	MoveL Offs(p0,623.8,790.0, 0), v100, z5, tool0;
	MoveL Offs(p0,621.6576000000002,788.0128000000002, 0), v100, z5, tool0;
	MoveL Offs(p0,619.9534,786.1551999999999, 0), v100, z5, tool0;
	MoveL Offs(p0,617.8928,783.7984, 0), v100, z5, tool0;
	MoveL Offs(p0,615.525,781.0, 0), v100, z5, tool0;
	MoveL Offs(p0,612.8992000000001,777.8176, 0), v100, z5, tool0;
	MoveL Offs(p0,610.0645999999999,774.3088, 0), v100, z5, tool0;
	MoveL Offs(p0,607.0704000000001,770.5312, 0), v100, z5, tool0;
	MoveL Offs(p0,603.9658,766.5424, 0), v100, z5, tool0;
	MoveL Offs(p0,600.8,762.4, 0), v100, z5, tool0;
	MoveL Offs(p0,596.1566,756.2386000000001, 0), v100, z5, tool0;
	MoveL Offs(p0,592.2368000000002,751.1248000000003, 0), v100, z5, tool0;
	MoveL Offs(p0,588.9361999999999,746.9541999999999, 0), v100, z5, tool0;
	MoveL Offs(p0,586.1504000000001,743.6224, 0), v100, z5, tool0;
	MoveL Offs(p0,583.775,741.025, 0), v100, z5, tool0;
	MoveL Offs(p0,581.7056,739.0576, 0), v100, z5, tool0;
	MoveL Offs(p0,579.8378,737.6157999999999, 0), v100, z5, tool0;
	MoveL Offs(p0,578.0672000000001,736.5952000000001, 0), v100, z5, tool0;
	MoveL Offs(p0,576.2894,735.8914000000001, 0), v100, z5, tool0;
	MoveL Offs(p0,574.4,735.4, 0), v100, z5, tool0;
	MoveL Offs(p0,566.3782000000001,733.9154000000001, 0), v100, z5, tool0;
	MoveL Offs(p0,559.1856000000001,732.8352000000002, 0), v100, z5, tool0;
	MoveL Offs(p0,552.5713999999999,732.1798000000001, 0), v100, z5, tool0;
	MoveL Offs(p0,546.2848,731.9696, 0), v100, z5, tool0;
	MoveL Offs(p0,540.075,732.225, 0), v100, z5, tool0;
	MoveL Offs(p0,533.6912,732.9664, 0), v100, z5, tool0;
	MoveL Offs(p0,526.8826,734.2142, 0), v100, z5, tool0;
	MoveL Offs(p0,519.3984,735.9888000000001, 0), v100, z5, tool0;
	MoveL Offs(p0,510.98780000000005,738.3106, 0), v100, z5, tool0;
	MoveL Offs(p0,501.4,741.2, 0), v100, z5, tool0;
	MoveL Offs(p0,496.9594000000001,742.5744000000001, 0), v100, z5, tool0;
	MoveL Offs(p0,492.63520000000017,743.8192000000001, 0), v100, z5, tool0;
	MoveL Offs(p0,488.4237999999999,744.9368, 0), v100, z5, tool0;
	MoveL Offs(p0,484.32159999999993,745.9296, 0), v100, z5, tool0;
	MoveL Offs(p0,480.325,746.8, 0), v100, z5, tool0;
	MoveL Offs(p0,476.4304,747.5504, 0), v100, z5, tool0;
	MoveL Offs(p0,472.63419999999996,748.1832, 0), v100, z5, tool0;
	MoveL Offs(p0,468.93280000000004,748.7008000000001, 0), v100, z5, tool0;
	MoveL Offs(p0,465.3226000000001,749.1056000000001, 0), v100, z5, tool0;
	MoveL Offs(p0,461.8,749.4, 0), v100, z5, tool0;
	MoveL Offs(p0,444.6,750.6, 0), v100, z5, tool0;
	MoveL Offs(p0,443.2,768.8, 0), v100, z5, tool0;
	MoveL Offs(p0,442.5474000000001,776.1014, 0), v100, z5, tool0;
	MoveL Offs(p0,441.5792000000001,784.0592000000003, 0), v100, z5, tool0;
	MoveL Offs(p0,440.3398,792.4538000000001, 0), v100, z5, tool0;
	MoveL Offs(p0,438.87360000000007,801.0656000000001, 0), v100, z5, tool0;
	MoveL Offs(p0,437.225,809.675, 0), v100, z5, tool0;
	MoveL Offs(p0,435.4384,818.0624, 0), v100, z5, tool0;
	MoveL Offs(p0,433.55820000000006,826.0082, 0), v100, z5, tool0;
	MoveL Offs(p0,431.62880000000007,833.2928000000002, 0), v100, z5, tool0;
	MoveL Offs(p0,429.6946,839.6966, 0), v100, z5, tool0;
	MoveL Offs(p0,427.8,845.0, 0), v100, z5, tool0;
	MoveL Offs(p0,426.53460000000007,848.1554, 0), v100, z5, tool0;
	MoveL Offs(p0,425.45280000000014,850.7072000000004, 0), v100, z5, tool0;
	MoveL Offs(p0,424.4862,852.7238, 0), v100, z5, tool0;
	MoveL Offs(p0,423.56640000000004,854.2736000000001, 0), v100, z5, tool0;
	MoveL Offs(p0,422.625,855.425, 0), v100, z5, tool0;
	MoveL Offs(p0,421.5936,856.2464, 0), v100, z5, tool0;
	MoveL Offs(p0,420.40380000000005,856.8062, 0), v100, z5, tool0;
	MoveL Offs(p0,418.98720000000003,857.1728, 0), v100, z5, tool0;
	MoveL Offs(p0,417.2754,857.4146000000001, 0), v100, z5, tool0;
	MoveL Offs(p0,415.2,857.6, 0), v100, z5, tool0;
	MoveL Offs(p0,407.4,858.2, 0), v100, z5, tool0;
	MoveL Offs(p0,408.8,838.6, 0), v100, z5, tool0;
	MoveL Offs(p0,410.0,819.0, 0), v100, z5, tool0;
	MoveL Offs(p0,403.8,834.0, 0), v100, z5, tool0;
	MoveL Offs(p0,400.23840000000007,842.4250000000002, 0), v100, z5, tool0;
	MoveL Offs(p0,396.2352000000001,851.4560000000004, 0), v100, z5, tool0;
	MoveL Offs(p0,391.9128,860.847, 0), v100, z5, tool0;
	MoveL Offs(p0,387.39360000000005,870.3520000000001, 0), v100, z5, tool0;
	MoveL Offs(p0,382.8,879.725, 0), v100, z5, tool0;
	MoveL Offs(p0,378.2544,888.72, 0), v100, z5, tool0;
	MoveL Offs(p0,373.8792,897.091, 0), v100, z5, tool0;
	MoveL Offs(p0,369.7968,904.5920000000002, 0), v100, z5, tool0;
	MoveL Offs(p0,366.12960000000004,910.9770000000001, 0), v100, z5, tool0;
	MoveL Offs(p0,363.0,916.0, 0), v100, z5, tool0;
	MoveL Offs(p0,359.5914000000001,920.9900000000001, 0), v100, z5, tool0;
	MoveL Offs(p0,356.51520000000005,925.2000000000004, 0), v100, z5, tool0;
	MoveL Offs(p0,353.6958,928.6899999999999, 0), v100, z5, tool0;
	MoveL Offs(p0,351.0576,931.5200000000001, 0), v100, z5, tool0;
	MoveL Offs(p0,348.525,933.75, 0), v100, z5, tool0;
	MoveL Offs(p0,346.0224,935.4399999999999, 0), v100, z5, tool0;
	MoveL Offs(p0,343.4742,936.65, 0), v100, z5, tool0;
	MoveL Offs(p0,340.8048,937.4400000000002, 0), v100, z5, tool0;
	MoveL Offs(p0,337.93860000000006,937.8700000000001, 0), v100, z5, tool0;
	MoveL Offs(p0,334.8,938.0, 0), v100, z5, tool0;
	MoveL Offs(p0,332.6582000000001,937.9793999999999, 0), v100, z5, tool0;
	MoveL Offs(p0,330.8896000000001,937.9072000000003, 0), v100, z5, tool0;
	MoveL Offs(p0,329.45939999999996,937.7678, 0), v100, z5, tool0;
	MoveL Offs(p0,328.3328,937.5456000000001, 0), v100, z5, tool0;
	MoveL Offs(p0,327.475,937.225, 0), v100, z5, tool0;
	MoveL Offs(p0,326.8512,936.7903999999999, 0), v100, z5, tool0;
	MoveL Offs(p0,326.4266,936.2262000000001, 0), v100, z5, tool0;
	MoveL Offs(p0,326.1664,935.5168000000001, 0), v100, z5, tool0;
	MoveL Offs(p0,326.0358,934.6466, 0), v100, z5, tool0;
	MoveL Offs(p0,326.0,933.6, 0), v100, z5, tool0;
	MoveL Offs(p0,326.0,933.6, 0), v100, z5, tool0;
	MoveJ Offs(p0,343.6,931.0, 10), v100, z1, tool0;
	MoveL Offs(p0,345.80180000000007,929.0856000000001, 0), v100, z5, tool0;
	MoveL Offs(p0,348.3984000000001,926.2928000000002, 0), v100, z5, tool0;
	MoveL Offs(p0,351.3166,922.7272, 0), v100, z5, tool0;
	MoveL Offs(p0,354.4832,918.4943999999999, 0), v100, z5, tool0;
	MoveL Offs(p0,357.825,913.7, 0), v100, z5, tool0;
	MoveL Offs(p0,361.2688,908.4495999999999, 0), v100, z5, tool0;
	MoveL Offs(p0,364.7414,902.8488, 0), v100, z5, tool0;
	MoveL Offs(p0,368.16960000000006,897.0031999999999, 0), v100, z5, tool0;
	MoveL Offs(p0,371.4802,891.0184000000002, 0), v100, z5, tool0;
	MoveL Offs(p0,374.6,885.0, 0), v100, z5, tool0;
	MoveL Offs(p0,379.89200000000005,873.9975999999999, 0), v100, z5, tool0;
	MoveL Offs(p0,385.01600000000013,862.6688000000001, 0), v100, z5, tool0;
	MoveL Offs(p0,389.864,851.3111999999999, 0), v100, z5, tool0;
	MoveL Offs(p0,394.32800000000003,840.2224, 0), v100, z5, tool0;
	MoveL Offs(p0,398.3,829.7, 0), v100, z5, tool0;
	MoveL Offs(p0,401.67199999999997,820.0415999999999, 0), v100, z5, tool0;
	MoveL Offs(p0,404.33599999999996,811.5448, 0), v100, z5, tool0;
	MoveL Offs(p0,406.184,804.5072, 0), v100, z5, tool0;
	MoveL Offs(p0,407.108,799.2264000000001, 0), v100, z5, tool0;
	MoveL Offs(p0,407.0,796.0, 0), v100, z5, tool0;
	MoveL Offs(p0,406.6202,793.9012, 0), v100, z5, tool0;
	MoveL Offs(p0,406.6544,793.3824000000002, 0), v100, z5, tool0;
	MoveL Offs(p0,406.775,792.95, 0), v100, z5, tool0;
	MoveL Offs(p0,406.9856,792.6016, 0), v100, z5, tool0;
	MoveL Offs(p0,407.2898,792.3348, 0), v100, z5, tool0;
	MoveL Offs(p0,407.69120000000004,792.1472000000001, 0), v100, z5, tool0;
	MoveL Offs(p0,408.1934,792.0364, 0), v100, z5, tool0;
	MoveL Offs(p0,408.8,792.0, 0), v100, z5, tool0;
	MoveL Offs(p0,411.23840000000007,793.0176000000001, 0), v100, z5, tool0;
	MoveL Offs(p0,412.1426,794.4084, 0), v100, z5, tool0;
	MoveL Offs(p0,412.85120000000006,796.4928, 0), v100, z5, tool0;
	MoveL Offs(p0,413.375,799.35, 0), v100, z5, tool0;
	MoveL Offs(p0,413.72479999999996,803.0592, 0), v100, z5, tool0;
	MoveL Offs(p0,413.91139999999996,807.6996, 0), v100, z5, tool0;
	MoveL Offs(p0,413.9456,813.3504, 0), v100, z5, tool0;
	MoveL Offs(p0,413.8382,820.0908, 0), v100, z5, tool0;
	MoveL Offs(p0,413.6,828.0, 0), v100, z5, tool0;
	MoveL Offs(p0,413.4460000000001,834.4142000000002, 0), v100, z5, tool0;
	MoveL Offs(p0,413.35200000000015,839.6896000000003, 0), v100, z5, tool0;
	MoveL Offs(p0,413.3299999999999,843.9354, 0), v100, z5, tool0;
	MoveL Offs(p0,413.392,847.2608, 0), v100, z5, tool0;
	MoveL Offs(p0,413.55,849.775, 0), v100, z5, tool0;
	MoveL Offs(p0,413.816,851.5871999999999, 0), v100, z5, tool0;
	MoveL Offs(p0,414.20200000000006,852.8066000000001, 0), v100, z5, tool0;
	MoveL Offs(p0,414.7200000000001,853.5424, 0), v100, z5, tool0;
	MoveL Offs(p0,415.38199999999995,853.9038, 0), v100, z5, tool0;
	MoveL Offs(p0,416.2,854.0, 0), v100, z5, tool0;
	MoveL Offs(p0,418.8432000000001,852.6416000000002, 0), v100, z5, tool0;
	MoveL Offs(p0,420.1708,850.9273999999999, 0), v100, z5, tool0;
	MoveL Offs(p0,421.5056000000001,848.5088, 0), v100, z5, tool0;
	MoveL Offs(p0,422.85,845.375, 0), v100, z5, tool0;
	MoveL Offs(p0,424.20640000000003,841.5152, 0), v100, z5, tool0;
	MoveL Offs(p0,425.5772,836.9186, 0), v100, z5, tool0;
	MoveL Offs(p0,426.9648,831.5744000000001, 0), v100, z5, tool0;
	MoveL Offs(p0,428.37160000000006,825.4718, 0), v100, z5, tool0;
	MoveL Offs(p0,429.8,818.6, 0), v100, z5, tool0;
	MoveL Offs(p0,431.0768,811.6862000000002, 0), v100, z5, tool0;
	MoveL Offs(p0,432.3584000000002,803.8976000000001, 0), v100, z5, tool0;
	MoveL Offs(p0,433.60159999999996,795.5834, 0), v100, z5, tool0;
	MoveL Offs(p0,434.76320000000004,787.0928000000001, 0), v100, z5, tool0;
	MoveL Offs(p0,435.8,778.775, 0), v100, z5, tool0;
	MoveL Offs(p0,436.66880000000003,770.9792, 0), v100, z5, tool0;
	MoveL Offs(p0,437.3263999999999,764.0546, 0), v100, z5, tool0;
	MoveL Offs(p0,437.7296,758.3504, 0), v100, z5, tool0;
	MoveL Offs(p0,437.8352,754.2158000000001, 0), v100, z5, tool0;
	MoveL Offs(p0,437.6,752.0, 0), v100, z5, tool0;
	MoveL Offs(p0,434.5075999999999,754.5325999999999, 0), v100, z5, tool0;
	MoveL Offs(p0,432.4032,756.8192, 0), v100, z5, tool0;
	MoveL Offs(p0,429.85,759.725, 0), v100, z5, tool0;
	MoveL Offs(p0,426.9008,763.1888, 0), v100, z5, tool0;
	MoveL Offs(p0,423.60839999999996,767.1494, 0), v100, z5, tool0;
	MoveL Offs(p0,420.02560000000005,771.5456000000001, 0), v100, z5, tool0;
	MoveL Offs(p0,416.20520000000005,776.3162, 0), v100, z5, tool0;
	MoveL Offs(p0,412.2,781.4, 0), v100, z5, tool0;
	MoveL Offs(p0,404.0998000000001,791.6810000000002, 0), v100, z5, tool0;
	MoveL Offs(p0,397.3424000000001,800.1920000000002, 0), v100, z5, tool0;
	MoveL Offs(p0,391.7826,807.095, 0), v100, z5, tool0;
	MoveL Offs(p0,387.27520000000004,812.552, 0), v100, z5, tool0;
	MoveL Offs(p0,383.675,816.725, 0), v100, z5, tool0;
	MoveL Offs(p0,380.8368,819.7759999999998, 0), v100, z5, tool0;
	MoveL Offs(p0,378.6154,821.867, 0), v100, z5, tool0;
	MoveL Offs(p0,376.86560000000003,823.1600000000001, 0), v100, z5, tool0;
	MoveL Offs(p0,375.4422,823.817, 0), v100, z5, tool0;
	MoveL Offs(p0,374.2,824.0, 0), v100, z5, tool0;
	MoveL Offs(p0,371.75680000000006,823.3696000000002, 0), v100, z5, tool0;
	MoveL Offs(p0,370.4092,822.6554, 0), v100, z5, tool0;
	MoveL Offs(p0,369.05440000000004,821.7408000000001, 0), v100, z5, tool0;
	MoveL Offs(p0,367.75,820.675, 0), v100, z5, tool0;
	MoveL Offs(p0,366.55359999999996,819.5072, 0), v100, z5, tool0;
	MoveL Offs(p0,365.5228,818.2866, 0), v100, z5, tool0;
	MoveL Offs(p0,364.7152,817.0624, 0), v100, z5, tool0;
	MoveL Offs(p0,364.1884,815.8838, 0), v100, z5, tool0;
	MoveL Offs(p0,364.0,814.8, 0), v100, z5, tool0;
	MoveL Offs(p0,364.86880000000014,811.4400000000002, 0), v100, z5, tool0;
	MoveL Offs(p0,366.0412,808.4010000000001, 0), v100, z5, tool0;
	MoveL Offs(p0,367.78240000000005,804.2880000000001, 0), v100, z5, tool0;
	MoveL Offs(p0,370.15,798.975, 0), v100, z5, tool0;
	MoveL Offs(p0,373.2016,792.336, 0), v100, z5, tool0;
	MoveL Offs(p0,376.99480000000005,784.2449999999999, 0), v100, z5, tool0;
	MoveL Offs(p0,381.58720000000005,774.576, 0), v100, z5, tool0;
	MoveL Offs(p0,387.03640000000007,763.2030000000001, 0), v100, z5, tool0;
	MoveL Offs(p0,393.4,750.0, 0), v100, z5, tool0;
	MoveL Offs(p0,399.2522000000001,737.9830000000001, 0), v100, z5, tool0;
	MoveL Offs(p0,404.2416000000001,727.6640000000003, 0), v100, z5, tool0;
	MoveL Offs(p0,408.4174,718.9409999999999, 0), v100, z5, tool0;
	MoveL Offs(p0,411.82880000000006,711.712, 0), v100, z5, tool0;
	MoveL Offs(p0,414.525,705.875, 0), v100, z5, tool0;
	MoveL Offs(p0,416.55519999999996,701.328, 0), v100, z5, tool0;
	MoveL Offs(p0,417.9686,697.9689999999998, 0), v100, z5, tool0;
	MoveL Offs(p0,418.81440000000003,695.6960000000001, 0), v100, z5, tool0;
	MoveL Offs(p0,419.1418,694.4069999999999, 0), v100, z5, tool0;
	MoveL Offs(p0,419.0,694.0, 0), v100, z5, tool0;
	MoveL Offs(p0,416.744,695.2864, 0), v100, z5, tool0;
	MoveL Offs(p0,415.775,695.95, 0), v100, z5, tool0;
	MoveL Offs(p0,414.68,696.7216000000001, 0), v100, z5, tool0;
	MoveL Offs(p0,413.477,697.5868, 0), v100, z5, tool0;
	MoveL Offs(p0,412.184,698.5312000000001, 0), v100, z5, tool0;
	MoveL Offs(p0,410.8190000000001,699.5404000000001, 0), v100, z5, tool0;
	MoveL Offs(p0,409.4,700.6, 0), v100, z5, tool0;
	MoveL Offs(p0,407.0394,702.3206000000001, 0), v100, z5, tool0;
	MoveL Offs(p0,404.53120000000007,703.9968000000002, 0), v100, z5, tool0;
	MoveL Offs(p0,401.8958,705.6202, 0), v100, z5, tool0;
	MoveL Offs(p0,399.1536,707.1823999999999, 0), v100, z5, tool0;
	MoveL Offs(p0,396.325,708.675, 0), v100, z5, tool0;
	MoveL Offs(p0,393.4304,710.0896, 0), v100, z5, tool0;
	MoveL Offs(p0,390.4902,711.4177999999999, 0), v100, z5, tool0;
	MoveL Offs(p0,387.5248,712.6512, 0), v100, z5, tool0;
	MoveL Offs(p0,384.55460000000005,713.7814000000001, 0), v100, z5, tool0;
	MoveL Offs(p0,381.6,714.8, 0), v100, z5, tool0;
	MoveL Offs(p0,379.2384,716.9222000000001, 0), v100, z5, tool0;
	MoveL Offs(p0,378.25280000000004,718.2464, 0), v100, z5, tool0;
	MoveL Offs(p0,377.2,719.825, 0), v100, z5, tool0;
	MoveL Offs(p0,376.0992,721.6256, 0), v100, z5, tool0;
	MoveL Offs(p0,374.9696,723.6157999999999, 0), v100, z5, tool0;
	MoveL Offs(p0,373.8304,725.7632000000001, 0), v100, z5, tool0;
	MoveL Offs(p0,372.7008,728.0354, 0), v100, z5, tool0;
	MoveL Offs(p0,371.6,730.4, 0), v100, z5, tool0;
	MoveL Offs(p0,368.85980000000006,736.4426000000001, 0), v100, z5, tool0;
	MoveL Offs(p0,366.1184000000001,742.2848000000002, 0), v100, z5, tool0;
	MoveL Offs(p0,363.31460000000004,748.0381999999998, 0), v100, z5, tool0;
	MoveL Offs(p0,360.3872,753.8144, 0), v100, z5, tool0;
	MoveL Offs(p0,357.275,759.725, 0), v100, z5, tool0;
	MoveL Offs(p0,353.91679999999997,765.8816, 0), v100, z5, tool0;
	MoveL Offs(p0,350.2514,772.3958, 0), v100, z5, tool0;
	MoveL Offs(p0,346.21760000000006,779.3792000000001, 0), v100, z5, tool0;
	MoveL Offs(p0,341.7542,786.9434, 0), v100, z5, tool0;
	MoveL Offs(p0,336.8,795.2, 0), v100, z5, tool0;
	MoveL Offs(p0,334.3450000000001,799.2708, 0), v100, z5, tool0;
	MoveL Offs(p0,332.0400000000001,803.1664000000003, 0), v100, z5, tool0;
	MoveL Offs(p0,329.91499999999996,806.8315999999999, 0), v100, z5, tool0;
	MoveL Offs(p0,328.0,810.2112000000001, 0), v100, z5, tool0;
	MoveL Offs(p0,326.325,813.25, 0), v100, z5, tool0;
	MoveL Offs(p0,324.91999999999996,815.8928, 0), v100, z5, tool0;
	MoveL Offs(p0,323.81499999999994,818.0844, 0), v100, z5, tool0;
	MoveL Offs(p0,323.0400000000001,819.7696, 0), v100, z5, tool0;
	MoveL Offs(p0,322.625,820.8932000000001, 0), v100, z5, tool0;
	MoveL Offs(p0,322.6,821.4, 0), v100, z5, tool0;
	MoveL Offs(p0,325.48900000000003,821.6735999999999, 0), v100, z5, tool0;
	MoveL Offs(p0,326.968,821.2592000000001, 0), v100, z5, tool0;
	MoveL Offs(p0,328.675,820.6, 0), v100, z5, tool0;
	MoveL Offs(p0,330.592,819.7008, 0), v100, z5, tool0;
	MoveL Offs(p0,332.701,818.5663999999999, 0), v100, z5, tool0;
	MoveL Offs(p0,334.98400000000004,817.2016000000001, 0), v100, z5, tool0;
	MoveL Offs(p0,337.42300000000006,815.6112, 0), v100, z5, tool0;
	MoveL Offs(p0,340.0,813.8, 0), v100, z5, tool0;
	MoveL Offs(p0,343.2048000000001,811.3024000000003, 0), v100, z5, tool0;
	MoveL Offs(p0,344.4352,810.2216, 0), v100, z5, tool0;
	MoveL Offs(p0,345.4304000000001,809.2272000000002, 0), v100, z5, tool0;
	MoveL Offs(p0,346.2,808.3, 0), v100, z5, tool0;
	MoveL Offs(p0,346.7536,807.4207999999999, 0), v100, z5, tool0;
	MoveL Offs(p0,347.1008,806.5704, 0), v100, z5, tool0;
	MoveL Offs(p0,347.25120000000004,805.7296000000001, 0), v100, z5, tool0;
	MoveL Offs(p0,347.21439999999996,804.8792000000001, 0), v100, z5, tool0;
	MoveL Offs(p0,347.0,804.0, 0), v100, z5, tool0;
	MoveL Offs(p0,346.5536,801.8129999999999, 0), v100, z5, tool0;
	MoveL Offs(p0,346.61920000000003,801.296, 0), v100, z5, tool0;
	MoveL Offs(p0,346.8,800.875, 0), v100, z5, tool0;
	MoveL Offs(p0,347.1008,800.544, 0), v100, z5, tool0;
	MoveL Offs(p0,347.5264,800.2969999999999, 0), v100, z5, tool0;
	MoveL Offs(p0,348.08160000000004,800.128, 0), v100, z5, tool0;
	MoveL Offs(p0,348.7712,800.0310000000001, 0), v100, z5, tool0;
	MoveL Offs(p0,349.6,800.0, 0), v100, z5, tool0;
	MoveL Offs(p0,351.7186,800.4752000000001, 0), v100, z5, tool0;
	MoveL Offs(p0,352.3232,800.8384, 0), v100, z5, tool0;
	MoveL Offs(p0,352.875,801.3, 0), v100, z5, tool0;
	MoveL Offs(p0,353.3728,801.8576, 0), v100, z5, tool0;
	MoveL Offs(p0,353.8154,802.5088, 0), v100, z5, tool0;
	MoveL Offs(p0,354.20160000000004,803.2512, 0), v100, z5, tool0;
	MoveL Offs(p0,354.53020000000004,804.0824, 0), v100, z5, tool0;
	MoveL Offs(p0,354.8,805.0, 0), v100, z5, tool0;
	MoveL Offs(p0,355.23800000000006,810.7434000000001, 0), v100, z5, tool0;
	MoveL Offs(p0,354.7280000000002,819.8912000000003, 0), v100, z5, tool0;
	MoveL Offs(p0,353.414,831.6598, 0), v100, z5, tool0;
	MoveL Offs(p0,351.44,845.2656000000001, 0), v100, z5, tool0;
	MoveL Offs(p0,348.95,859.925, 0), v100, z5, tool0;
	MoveL Offs(p0,346.08799999999997,874.8543999999999, 0), v100, z5, tool0;
	MoveL Offs(p0,342.998,889.2702000000002, 0), v100, z5, tool0;
	MoveL Offs(p0,339.82400000000007,902.3888000000001, 0), v100, z5, tool0;
	MoveL Offs(p0,336.71000000000004,913.4266, 0), v100, z5, tool0;
	MoveL Offs(p0,333.8,921.6, 0), v100, z5, tool0;
	MoveL Offs(p0,332.5600000000001,924.4496000000003, 0), v100, z5, tool0;
	MoveL Offs(p0,332.00899999999996,925.8173999999999, 0), v100, z5, tool0;
	MoveL Offs(p0,331.512,927.1168000000001, 0), v100, z5, tool0;
	MoveL Offs(p0,331.075,928.325, 0), v100, z5, tool0;
	MoveL Offs(p0,330.704,929.4192, 0), v100, z5, tool0;
	MoveL Offs(p0,330.40500000000003,930.3765999999999, 0), v100, z5, tool0;
	MoveL Offs(p0,330.184,931.1744000000001, 0), v100, z5, tool0;
	MoveL Offs(p0,330.047,931.7898000000001, 0), v100, z5, tool0;
	MoveL Offs(p0,330.0,932.2, 0), v100, z5, tool0;
	MoveL Offs(p0,333.34720000000004,933.9087999999999, 0), v100, z5, tool0;
	MoveL Offs(p0,334.925,933.85, 0), v100, z5, tool0;
	MoveL Offs(p0,336.6528,933.6112, 0), v100, z5, tool0;
	MoveL Offs(p0,338.4574,933.1995999999999, 0), v100, z5, tool0;
	MoveL Offs(p0,340.2656,932.6224000000002, 0), v100, z5, tool0;
	MoveL Offs(p0,342.0042,931.8868, 0), v100, z5, tool0;
	MoveL Offs(p0,343.6,931.0, 0), v100, z5, tool0;
	MoveL Offs(p0,343.6,931.0, 0), v100, z5, tool0;
	MoveJ Offs(p0,252.4,787.0, 10), v100, z1, tool0;
	MoveL Offs(p0,254.81320000000005,785.7228000000001, 0), v100, z5, tool0;
	MoveL Offs(p0,257.56960000000004,784.1984000000001, 0), v100, z5, tool0;
	MoveL Offs(p0,260.6044,782.4675999999998, 0), v100, z5, tool0;
	MoveL Offs(p0,263.8528,780.5712000000001, 0), v100, z5, tool0;
	MoveL Offs(p0,267.25,778.55, 0), v100, z5, tool0;
	MoveL Offs(p0,270.7312,776.4448, 0), v100, z5, tool0;
	MoveL Offs(p0,274.23159999999996,774.2964, 0), v100, z5, tool0;
	MoveL Offs(p0,277.68640000000005,772.1456000000001, 0), v100, z5, tool0;
	MoveL Offs(p0,281.0308,770.0332000000001, 0), v100, z5, tool0;
	MoveL Offs(p0,284.2,768.0, 0), v100, z5, tool0;
	MoveL Offs(p0,288.2024,765.2460000000002, 0), v100, z5, tool0;
	MoveL Offs(p0,291.5952000000001,762.8400000000001, 0), v100, z5, tool0;
	MoveL Offs(p0,294.4168,760.7459999999999, 0), v100, z5, tool0;
	MoveL Offs(p0,296.70560000000006,758.9280000000001, 0), v100, z5, tool0;
	MoveL Offs(p0,298.5,757.35, 0), v100, z5, tool0;
	MoveL Offs(p0,299.8384,755.976, 0), v100, z5, tool0;
	MoveL Offs(p0,300.75919999999996,754.7700000000001, 0), v100, z5, tool0;
	MoveL Offs(p0,301.30080000000004,753.6960000000001, 0), v100, z5, tool0;
	MoveL Offs(p0,301.5016,752.7180000000001, 0), v100, z5, tool0;
	MoveL Offs(p0,301.4,751.8, 0), v100, z5, tool0;
	MoveL Offs(p0,301.1792000000001,749.7504000000001, 0), v100, z5, tool0;
	MoveL Offs(p0,301.3208,749.0046, 0), v100, z5, tool0;
	MoveL Offs(p0,301.60159999999996,748.4592, 0), v100, z5, tool0;
	MoveL Offs(p0,302.0,748.125, 0), v100, z5, tool0;
	MoveL Offs(p0,302.4944,748.0128, 0), v100, z5, tool0;
	MoveL Offs(p0,303.06319999999994,748.1333999999999, 0), v100, z5, tool0;
	MoveL Offs(p0,303.6848,748.4976, 0), v100, z5, tool0;
	MoveL Offs(p0,304.3376,749.1162, 0), v100, z5, tool0;
	MoveL Offs(p0,305.0,750.0, 0), v100, z5, tool0;
	MoveL Offs(p0,305.2699999999999,752.3202, 0), v100, z5, tool0;
	MoveL Offs(p0,305.24000000000007,753.6384, 0), v100, z5, tool0;
	MoveL Offs(p0,305.15,755.175, 0), v100, z5, tool0;
	MoveL Offs(p0,305.0,756.8976, 0), v100, z5, tool0;
	MoveL Offs(p0,304.78999999999996,758.7738, 0), v100, z5, tool0;
	MoveL Offs(p0,304.52000000000004,760.7712000000001, 0), v100, z5, tool0;
	MoveL Offs(p0,304.19,762.8574000000001, 0), v100, z5, tool0;
	MoveL Offs(p0,303.8,765.0, 0), v100, z5, tool0;
	MoveL Offs(p0,303.4642,767.1366, 0), v100, z5, tool0;
	MoveL Offs(p0,303.1776000000001,769.2048000000002, 0), v100, z5, tool0;
	MoveL Offs(p0,302.94140000000004,771.1722, 0), v100, z5, tool0;
	MoveL Offs(p0,302.7568,773.0064, 0), v100, z5, tool0;
	MoveL Offs(p0,302.625,774.675, 0), v100, z5, tool0;
	MoveL Offs(p0,302.5472,776.1456000000001, 0), v100, z5, tool0;
	MoveL Offs(p0,302.5246,777.3858, 0), v100, z5, tool0;
	MoveL Offs(p0,302.55840000000006,778.3632000000001, 0), v100, z5, tool0;
	MoveL Offs(p0,302.6498,779.0454000000001, 0), v100, z5, tool0;
	MoveL Offs(p0,302.8,779.4, 0), v100, z5, tool0;
	MoveL Offs(p0,307.29600000000016,777.1200000000002, 0), v100, z5, tool0;
	MoveL Offs(p0,311.16999999999996,773.406, 0), v100, z5, tool0;
	MoveL Offs(p0,315.776,768.4080000000001, 0), v100, z5, tool0;
	MoveL Offs(p0,320.85,762.45, 0), v100, z5, tool0;
	MoveL Offs(p0,326.12800000000004,755.856, 0), v100, z5, tool0;
	MoveL Offs(p0,331.346,748.95, 0), v100, z5, tool0;
	MoveL Offs(p0,336.24000000000007,742.0560000000002, 0), v100, z5, tool0;
	MoveL Offs(p0,340.546,735.498, 0), v100, z5, tool0;
	MoveL Offs(p0,344.0,729.6, 0), v100, z5, tool0;
	MoveL Offs(p0,348.6,720.6, 0), v100, z5, tool0;
	MoveL Offs(p0,332.8,705.2, 0), v100, z5, tool0;
	MoveL Offs(p0,329.8550000000001,702.4052, 0), v100, z5, tool0;
	MoveL Offs(p0,327.1440000000001,699.9056000000002, 0), v100, z5, tool0;
	MoveL Offs(p0,324.67299999999994,697.7083999999999, 0), v100, z5, tool0;
	MoveL Offs(p0,322.448,695.8208, 0), v100, z5, tool0;
	MoveL Offs(p0,320.475,694.25, 0), v100, z5, tool0;
	MoveL Offs(p0,318.75999999999993,693.0031999999999, 0), v100, z5, tool0;
	MoveL Offs(p0,317.309,692.0876000000001, 0), v100, z5, tool0;
	MoveL Offs(p0,316.12800000000004,691.5104, 0), v100, z5, tool0;
	MoveL Offs(p0,315.223,691.2788, 0), v100, z5, tool0;
	MoveL Offs(p0,314.6,691.4, 0), v100, z5, tool0;
	MoveL Offs(p0,305.2424,697.7650000000001, 0), v100, z5, tool0;
	MoveL Offs(p0,297.2672000000001,703.224, 0), v100, z5, tool0;
	MoveL Offs(p0,290.58079999999995,707.843, 0), v100, z5, tool0;
	MoveL Offs(p0,285.0896,711.6880000000001, 0), v100, z5, tool0;
	MoveL Offs(p0,280.7,714.825, 0), v100, z5, tool0;
	MoveL Offs(p0,277.3184,717.3199999999999, 0), v100, z5, tool0;
	MoveL Offs(p0,274.85119999999995,719.239, 0), v100, z5, tool0;
	MoveL Offs(p0,273.20480000000003,720.648, 0), v100, z5, tool0;
	MoveL Offs(p0,272.28560000000004,721.613, 0), v100, z5, tool0;
	MoveL Offs(p0,272.0,722.2, 0), v100, z5, tool0;
	MoveL Offs(p0,274.35,723.475, 0), v100, z5, tool0;
	MoveL Offs(p0,275.28319999999997,723.6544, 0), v100, z5, tool0;
	MoveL Offs(p0,276.3316,723.8002, 0), v100, z5, tool0;
	MoveL Offs(p0,277.4784000000001,723.9088, 0), v100, z5, tool0;
	MoveL Offs(p0,278.70680000000004,723.9766000000001, 0), v100, z5, tool0;
	MoveL Offs(p0,280.0,724.0, 0), v100, z5, tool0;
	MoveL Offs(p0,282.14400000000006,723.9252000000001, 0), v100, z5, tool0;
	MoveL Offs(p0,284.00000000000006,723.7136000000002, 0), v100, z5, tool0;
	MoveL Offs(p0,285.544,723.3844, 0), v100, z5, tool0;
	MoveL Offs(p0,286.75200000000007,722.9568, 0), v100, z5, tool0;
	MoveL Offs(p0,287.6,722.45, 0), v100, z5, tool0;
	MoveL Offs(p0,288.06399999999996,721.8832, 0), v100, z5, tool0;
	MoveL Offs(p0,288.12,721.2755999999999, 0), v100, z5, tool0;
	MoveL Offs(p0,287.744,720.6464, 0), v100, z5, tool0;
	MoveL Offs(p0,286.91200000000003,720.0148, 0), v100, z5, tool0;
	MoveL Offs(p0,285.6,719.4, 0), v100, z5, tool0;
	MoveL Offs(p0,288.94080000000014,718.4800000000002, 0), v100, z5, tool0;
	MoveL Offs(p0,289.8632,718.911, 0), v100, z5, tool0;
	MoveL Offs(p0,290.5504,719.528, 0), v100, z5, tool0;
	MoveL Offs(p0,291.0,720.325, 0), v100, z5, tool0;
	MoveL Offs(p0,291.20959999999997,721.2959999999999, 0), v100, z5, tool0;
	MoveL Offs(p0,291.1768,722.4350000000001, 0), v100, z5, tool0;
	MoveL Offs(p0,290.8992,723.7360000000001, 0), v100, z5, tool0;
	MoveL Offs(p0,290.37440000000004,725.193, 0), v100, z5, tool0;
	MoveL Offs(p0,289.6,726.8, 0), v100, z5, tool0;
	MoveL Offs(p0,286.4896000000001,731.2496000000001, 0), v100, z5, tool0;
	MoveL Offs(p0,283.8094,734.6084, 0), v100, z5, tool0;
	MoveL Offs(p0,280.4128,738.6848000000001, 0), v100, z5, tool0;
	MoveL Offs(p0,276.325,743.45, 0), v100, z5, tool0;
	MoveL Offs(p0,271.5712,748.8752, 0), v100, z5, tool0;
	MoveL Offs(p0,266.17659999999995,754.9316000000001, 0), v100, z5, tool0;
	MoveL Offs(p0,260.1664,761.5904, 0), v100, z5, tool0;
	MoveL Offs(p0,253.56580000000002,768.8228, 0), v100, z5, tool0;
	MoveL Offs(p0,246.4,776.6, 0), v100, z5, tool0;
	MoveL Offs(p0,243.34560000000005,779.9060000000001, 0), v100, z5, tool0;
	MoveL Offs(p0,240.78080000000006,782.8640000000003, 0), v100, z5, tool0;
	MoveL Offs(p0,238.7032,785.4739999999999, 0), v100, z5, tool0;
	MoveL Offs(p0,237.11039999999997,787.736, 0), v100, z5, tool0;
	MoveL Offs(p0,236.0,789.65, 0), v100, z5, tool0;
	MoveL Offs(p0,235.3696,791.216, 0), v100, z5, tool0;
	MoveL Offs(p0,235.2168,792.434, 0), v100, z5, tool0;
	MoveL Offs(p0,235.53920000000002,793.3040000000001, 0), v100, z5, tool0;
	MoveL Offs(p0,236.33440000000002,793.826, 0), v100, z5, tool0;
	MoveL Offs(p0,237.6,794.0, 0), v100, z5, tool0;
	MoveL Offs(p0,239.75100000000003,793.2061999999999, 0), v100, z5, tool0;
	MoveL Offs(p0,241.02400000000003,792.6304, 0), v100, z5, tool0;
	MoveL Offs(p0,242.525,791.925, 0), v100, z5, tool0;
	MoveL Offs(p0,244.22400000000002,791.1056, 0), v100, z5, tool0;
	MoveL Offs(p0,246.09099999999998,790.1877999999999, 0), v100, z5, tool0;
	MoveL Offs(p0,248.096,789.1872000000001, 0), v100, z5, tool0;
	MoveL Offs(p0,250.209,788.1193999999999, 0), v100, z5, tool0;
	MoveL Offs(p0,252.4,787.0, 0), v100, z5, tool0;
	MoveL Offs(p0,252.4,787.0, 0), v100, z5, tool0;
	MoveJ Offs(p0,851.2,780.4, 10), v100, z1, tool0;
	MoveL Offs(p0,853.4733999999999,777.8494, 0), v100, z5, tool0;
	MoveL Offs(p0,854.0128000000001,776.7648000000002, 0), v100, z5, tool0;
	MoveL Offs(p0,854.425,775.625, 0), v100, z5, tool0;
	MoveL Offs(p0,854.6992,774.4672, 0), v100, z5, tool0;
	MoveL Offs(p0,854.8245999999999,773.3285999999999, 0), v100, z5, tool0;
	MoveL Offs(p0,854.7904000000001,772.2464, 0), v100, z5, tool0;
	MoveL Offs(p0,854.5858000000001,771.2578, 0), v100, z5, tool0;
	MoveL Offs(p0,854.2,770.4, 0), v100, z5, tool0;
	MoveL Offs(p0,851.7573999999998,768.3048, 0), v100, z5, tool0;
	MoveL Offs(p0,850.2768,767.2256, 0), v100, z5, tool0;
	MoveL Offs(p0,848.525,766.0, 0), v100, z5, tool0;
	MoveL Offs(p0,846.5391999999999,764.6544, 0), v100, z5, tool0;
	MoveL Offs(p0,844.3565999999998,763.2152, 0), v100, z5, tool0;
	MoveL Offs(p0,842.0144,761.7088000000001, 0), v100, z5, tool0;
	MoveL Offs(p0,839.5498,760.1616, 0), v100, z5, tool0;
	MoveL Offs(p0,837.0,758.6, 0), v100, z5, tool0;
	MoveL Offs(p0,821.0282,748.1876, 0), v100, z5, tool0;
	MoveL Offs(p0,802.8976000000004,735.0368000000002, 0), v100, z5, tool0;
	MoveL Offs(p0,783.3653999999999,719.8172, 0), v100, z5, tool0;
	MoveL Offs(p0,763.1888000000001,703.1984, 0), v100, z5, tool0;
	MoveL Offs(p0,743.125,685.85, 0), v100, z5, tool0;
	MoveL Offs(p0,723.9312,668.4415999999999, 0), v100, z5, tool0;
	MoveL Offs(p0,706.3646,651.6428, 0), v100, z5, tool0;
	MoveL Offs(p0,691.1824,636.1232, 0), v100, z5, tool0;
	MoveL Offs(p0,679.1418000000001,622.5523999999999, 0), v100, z5, tool0;
	MoveL Offs(p0,671.0,611.6, 0), v100, z5, tool0;
	MoveL Offs(p0,668.9792000000001,608.6240000000001, 0), v100, z5, tool0;
	MoveL Offs(p0,668.0047999999999,607.271, 0), v100, z5, tool0;
	MoveL Offs(p0,667.0736,606.0319999999999, 0), v100, z5, tool0;
	MoveL Offs(p0,666.2,604.925, 0), v100, z5, tool0;
	MoveL Offs(p0,665.3984,603.968, 0), v100, z5, tool0;
	MoveL Offs(p0,664.6831999999999,603.179, 0), v100, z5, tool0;
	MoveL Offs(p0,664.0688,602.576, 0), v100, z5, tool0;
	MoveL Offs(p0,663.5696,602.177, 0), v100, z5, tool0;
	MoveL Offs(p0,663.2,602.0, 0), v100, z5, tool0;
	MoveL Offs(p0,662.325,604.75, 0), v100, z5, tool0;
	MoveL Offs(p0,662.3072,605.8448, 0), v100, z5, tool0;
	MoveL Offs(p0,662.3446,607.0763999999999, 0), v100, z5, tool0;
	MoveL Offs(p0,662.4384,608.4256000000001, 0), v100, z5, tool0;
	MoveL Offs(p0,662.5898000000001,609.8732, 0), v100, z5, tool0;
	MoveL Offs(p0,662.8,611.4, 0), v100, z5, tool0;
	MoveL Offs(p0,664.1762000000001,617.4388000000001, 0), v100, z5, tool0;
	MoveL Offs(p0,666.6576000000002,624.2624000000002, 0), v100, z5, tool0;
	MoveL Offs(p0,670.1134,631.6716, 0), v100, z5, tool0;
	MoveL Offs(p0,674.4128000000001,639.4672000000002, 0), v100, z5, tool0;
	MoveL Offs(p0,679.425,647.45, 0), v100, z5, tool0;
	MoveL Offs(p0,685.0192,655.4208, 0), v100, z5, tool0;
	MoveL Offs(p0,691.0646,663.1804, 0), v100, z5, tool0;
	MoveL Offs(p0,697.4304000000001,670.5296000000001, 0), v100, z5, tool0;
	MoveL Offs(p0,703.9858,677.2692, 0), v100, z5, tool0;
	MoveL Offs(p0,710.6,683.2, 0), v100, z5, tool0;
	MoveL Offs(p0,716.556,688.1088000000001, 0), v100, z5, tool0;
	MoveL Offs(p0,722.1520000000002,692.6144000000003, 0), v100, z5, tool0;
	MoveL Offs(p0,727.3399999999999,696.6856, 0), v100, z5, tool0;
	MoveL Offs(p0,732.0720000000001,700.2912, 0), v100, z5, tool0;
	MoveL Offs(p0,736.3,703.4, 0), v100, z5, tool0;
	MoveL Offs(p0,739.976,705.9808, 0), v100, z5, tool0;
	MoveL Offs(p0,743.052,708.0024000000001, 0), v100, z5, tool0;
	MoveL Offs(p0,745.4800000000001,709.4336000000001, 0), v100, z5, tool0;
	MoveL Offs(p0,747.2120000000001,710.2432000000001, 0), v100, z5, tool0;
	MoveL Offs(p0,748.2,710.4, 0), v100, z5, tool0;
	MoveL Offs(p0,750.6224000000002,714.1520000000002, 0), v100, z5, tool0;
	MoveL Offs(p0,752.0336,715.6699999999998, 0), v100, z5, tool0;
	MoveL Offs(p0,753.8432,717.2720000000002, 0), v100, z5, tool0;
	MoveL Offs(p0,755.9,718.85, 0), v100, z5, tool0;
	MoveL Offs(p0,758.0528,720.2959999999999, 0), v100, z5, tool0;
	MoveL Offs(p0,760.1504,721.5020000000001, 0), v100, z5, tool0;
	MoveL Offs(p0,762.0416000000001,722.36, 0), v100, z5, tool0;
	MoveL Offs(p0,763.5752,722.7620000000001, 0), v100, z5, tool0;
	MoveL Offs(p0,764.6,722.6, 0), v100, z5, tool0;
	MoveL Offs(p0,765.9360000000001,726.0288000000002, 0), v100, z5, tool0;
	MoveL Offs(p0,766.6,726.825, 0), v100, z5, tool0;
	MoveL Offs(p0,767.432,727.6752, 0), v100, z5, tool0;
	MoveL Offs(p0,768.42,728.5686, 0), v100, z5, tool0;
	MoveL Offs(p0,769.552,729.4944, 0), v100, z5, tool0;
	MoveL Offs(p0,770.816,730.4418000000001, 0), v100, z5, tool0;
	MoveL Offs(p0,772.2,731.4, 0), v100, z5, tool0;
	MoveL Offs(p0,774.9656000000001,733.2664000000002, 0), v100, z5, tool0;
	MoveL Offs(p0,777.4528000000003,734.9552000000002, 0), v100, z5, tool0;
	MoveL Offs(p0,779.7672,736.5408, 0), v100, z5, tool0;
	MoveL Offs(p0,782.0144,738.0976000000002, 0), v100, z5, tool0;
	MoveL Offs(p0,784.3,739.7, 0), v100, z5, tool0;
	MoveL Offs(p0,786.7295999999999,741.4223999999999, 0), v100, z5, tool0;
	MoveL Offs(p0,789.4087999999999,743.3392, 0), v100, z5, tool0;
	MoveL Offs(p0,792.4432,745.5248, 0), v100, z5, tool0;
	MoveL Offs(p0,795.9384,748.0536, 0), v100, z5, tool0;
	MoveL Offs(p0,800.0,751.0, 0), v100, z5, tool0;
	MoveL Offs(p0,803.5168000000002,753.4992000000002, 0), v100, z5, tool0;
	MoveL Offs(p0,805.1732,754.6197999999999, 0), v100, z5, tool0;
	MoveL Offs(p0,806.7264000000001,755.6336, 0), v100, z5, tool0;
	MoveL Offs(p0,808.15,756.525, 0), v100, z5, tool0;
	MoveL Offs(p0,809.4176,757.2783999999999, 0), v100, z5, tool0;
	MoveL Offs(p0,810.5028,757.8782, 0), v100, z5, tool0;
	MoveL Offs(p0,811.3792000000001,758.3088, 0), v100, z5, tool0;
	MoveL Offs(p0,812.0204,758.5546, 0), v100, z5, tool0;
	MoveL Offs(p0,812.4,758.6, 0), v100, z5, tool0;
	MoveL Offs(p0,817.2864000000003,762.8000000000002, 0), v100, z5, tool0;
	MoveL Offs(p0,820.8526000000002,765.389, 0), v100, z5, tool0;
	MoveL Offs(p0,825.2192000000001,768.392, 0), v100, z5, tool0;
	MoveL Offs(p0,830.025,771.575, 0), v100, z5, tool0;
	MoveL Offs(p0,834.9087999999999,774.704, 0), v100, z5, tool0;
	MoveL Offs(p0,839.5094000000001,777.5449999999998, 0), v100, z5, tool0;
	MoveL Offs(p0,843.4656000000001,779.8640000000001, 0), v100, z5, tool0;
	MoveL Offs(p0,846.4162,781.427, 0), v100, z5, tool0;
	MoveL Offs(p0,848.0,782.0, 0), v100, z5, tool0;
	MoveL Offs(p0,850.0930000000001,781.0984000000001, 0), v100, z5, tool0;
	MoveL Offs(p0,850.4639999999999,780.8736000000001, 0), v100, z5, tool0;
	MoveL Offs(p0,850.835,780.6392000000001, 0), v100, z5, tool0;
	MoveL Offs(p0,851.2,780.4, 0), v100, z5, tool0;
	MoveL Offs(p0,851.2,780.4, 0), v100, z5, tool0;
	MoveJ Offs(p0,830.0,739.8, 10), v100, z1, tool0;
	MoveL Offs(p0,827.7316000000001,732.0532000000001, 0), v100, z5, tool0;
	MoveL Offs(p0,826.0848000000002,724.0976000000003, 0), v100, z5, tool0;
	MoveL Offs(p0,825.0572,716.0004, 0), v100, z5, tool0;
	MoveL Offs(p0,824.6464,707.8288, 0), v100, z5, tool0;
	MoveL Offs(p0,824.85,699.65, 0), v100, z5, tool0;
	MoveL Offs(p0,825.6655999999999,691.5312, 0), v100, z5, tool0;
	MoveL Offs(p0,827.0908,683.5396, 0), v100, z5, tool0;
	MoveL Offs(p0,829.1232,675.7424000000001, 0), v100, z5, tool0;
	MoveL Offs(p0,831.7603999999999,668.2068, 0), v100, z5, tool0;
	MoveL Offs(p0,835.0,661.0, 0), v100, z5, tool0;
	MoveL Offs(p0,837.0346000000002,656.7876, 0), v100, z5, tool0;
	MoveL Offs(p0,838.7008000000002,653.0048000000002, 0), v100, z5, tool0;
	MoveL Offs(p0,840.0022000000001,649.6132, 0), v100, z5, tool0;
	MoveL Offs(p0,840.9424000000001,646.5744, 0), v100, z5, tool0;
	MoveL Offs(p0,841.525,643.85, 0), v100, z5, tool0;
	MoveL Offs(p0,841.7536,641.4016, 0), v100, z5, tool0;
	MoveL Offs(p0,841.6317999999999,639.1908, 0), v100, z5, tool0;
	MoveL Offs(p0,841.1632000000002,637.1792000000002, 0), v100, z5, tool0;
	MoveL Offs(p0,840.3514000000001,635.3284, 0), v100, z5, tool0;
	MoveL Offs(p0,839.2,633.6, 0), v100, z5, tool0;
	MoveL Offs(p0,835.2416000000001,630.2528000000001, 0), v100, z5, tool0;
	MoveL Offs(p0,832.0773999999999,628.3871999999999, 0), v100, z5, tool0;
	MoveL Offs(p0,828.2688,626.4544, 0), v100, z5, tool0;
	MoveL Offs(p0,823.925,624.5, 0), v100, z5, tool0;
	MoveL Offs(p0,819.1552,622.5696, 0), v100, z5, tool0;
	MoveL Offs(p0,814.0686,620.7088, 0), v100, z5, tool0;
	MoveL Offs(p0,808.7744,618.9632, 0), v100, z5, tool0;
	MoveL Offs(p0,803.3818000000001,617.3783999999999, 0), v100, z5, tool0;
	MoveL Offs(p0,798.0,616.0, 0), v100, z5, tool0;
	MoveL Offs(p0,788.8612,613.5534, 0), v100, z5, tool0;
	MoveL Offs(p0,779.5136000000002,610.6832000000002, 0), v100, z5, tool0;
	MoveL Offs(p0,770.0604,607.4338, 0), v100, z5, tool0;
	MoveL Offs(p0,760.6048000000001,603.8496000000001, 0), v100, z5, tool0;
	MoveL Offs(p0,751.25,599.975, 0), v100, z5, tool0;
	MoveL Offs(p0,742.0992,595.8543999999999, 0), v100, z5, tool0;
	MoveL Offs(p0,733.2556,591.5322, 0), v100, z5, tool0;
	MoveL Offs(p0,724.8224000000001,587.0528, 0), v100, z5, tool0;
	MoveL Offs(p0,716.9028000000001,582.4606, 0), v100, z5, tool0;
	MoveL Offs(p0,709.6,577.8, 0), v100, z5, tool0;
	MoveL Offs(p0,706.9404000000001,575.997, 0), v100, z5, tool0;
	MoveL Offs(p0,704.6912000000002,574.5360000000002, 0), v100, z5, tool0;
	MoveL Offs(p0,702.8068000000001,573.399, 0), v100, z5, tool0;
	MoveL Offs(p0,701.2416000000001,572.568, 0), v100, z5, tool0;
	MoveL Offs(p0,699.95,572.025, 0), v100, z5, tool0;
	MoveL Offs(p0,698.8864,571.752, 0), v100, z5, tool0;
	MoveL Offs(p0,698.0052,571.731, 0), v100, z5, tool0;
	MoveL Offs(p0,697.2608,571.9440000000001, 0), v100, z5, tool0;
	MoveL Offs(p0,696.6076,572.373, 0), v100, z5, tool0;
	MoveL Offs(p0,696.0,573.0, 0), v100, z5, tool0;
	MoveL Offs(p0,693.858,574.4418000000001, 0), v100, z5, tool0;
	MoveL Offs(p0,692.864,574.8336, 0), v100, z5, tool0;
	MoveL Offs(p0,691.75,575.175, 0), v100, z5, tool0;
	MoveL Offs(p0,690.528,575.4624000000001, 0), v100, z5, tool0;
	MoveL Offs(p0,689.2099999999999,575.6922, 0), v100, z5, tool0;
	MoveL Offs(p0,687.808,575.8608, 0), v100, z5, tool0;
	MoveL Offs(p0,686.3340000000001,575.9646, 0), v100, z5, tool0;
	MoveL Offs(p0,684.8,576.0, 0), v100, z5, tool0;
	MoveL Offs(p0,682.1534000000001,576.0766000000001, 0), v100, z5, tool0;
	MoveL Offs(p0,679.8272000000001,576.3248000000001, 0), v100, z5, tool0;
	MoveL Offs(p0,677.7818,576.7722, 0), v100, z5, tool0;
	MoveL Offs(p0,675.9776000000002,577.4464, 0), v100, z5, tool0;
	MoveL Offs(p0,674.375,578.375, 0), v100, z5, tool0;
	MoveL Offs(p0,672.9344,579.5856, 0), v100, z5, tool0;
	MoveL Offs(p0,671.6162,581.1058, 0), v100, z5, tool0;
	MoveL Offs(p0,670.3808000000001,582.9631999999999, 0), v100, z5, tool0;
	MoveL Offs(p0,669.1886000000001,585.1854000000001, 0), v100, z5, tool0;
	MoveL Offs(p0,668.0,587.8, 0), v100, z5, tool0;
	MoveL Offs(p0,666.9360000000003,590.8208000000001, 0), v100, z5, tool0;
	MoveL Offs(p0,666.731,592.1181999999999, 0), v100, z5, tool0;
	MoveL Offs(p0,666.784,593.3904, 0), v100, z5, tool0;
	MoveL Offs(p0,667.125,594.725, 0), v100, z5, tool0;
	MoveL Offs(p0,667.784,596.2095999999999, 0), v100, z5, tool0;
	MoveL Offs(p0,668.7909999999999,597.9318, 0), v100, z5, tool0;
	MoveL Offs(p0,670.176,599.9792, 0), v100, z5, tool0;
	MoveL Offs(p0,671.969,602.4394, 0), v100, z5, tool0;
	MoveL Offs(p0,674.2,605.4, 0), v100, z5, tool0;
	MoveL Offs(p0,681.1906,614.0184000000002, 0), v100, z5, tool0;
	MoveL Offs(p0,690.4768000000001,624.4752000000002, 0), v100, z5, tool0;
	MoveL Offs(p0,701.6302000000001,636.3527999999999, 0), v100, z5, tool0;
	MoveL Offs(p0,714.2224,649.2336, 0), v100, z5, tool0;
	MoveL Offs(p0,727.825,662.7, 0), v100, z5, tool0;
	MoveL Offs(p0,742.0096,676.3344, 0), v100, z5, tool0;
	MoveL Offs(p0,756.3478,689.7192000000001, 0), v100, z5, tool0;
	MoveL Offs(p0,770.4112000000001,702.4368000000001, 0), v100, z5, tool0;
	MoveL Offs(p0,783.7714000000001,714.0696, 0), v100, z5, tool0;
	MoveL Offs(p0,796.0,724.2, 0), v100, z5, tool0;
	MoveL Offs(p0,801.3996000000001,728.4282000000001, 0), v100, z5, tool0;
	MoveL Offs(p0,806.7248000000002,732.5376000000003, 0), v100, z5, tool0;
	MoveL Offs(p0,811.8652,736.4454, 0), v100, z5, tool0;
	MoveL Offs(p0,816.7104000000002,740.0688, 0), v100, z5, tool0;
	MoveL Offs(p0,821.15,743.325, 0), v100, z5, tool0;
	MoveL Offs(p0,825.0735999999999,746.1312, 0), v100, z5, tool0;
	MoveL Offs(p0,828.3707999999999,748.4046000000001, 0), v100, z5, tool0;
	MoveL Offs(p0,830.9312000000002,750.0624, 0), v100, z5, tool0;
	MoveL Offs(p0,832.6443999999999,751.0218, 0), v100, z5, tool0;
	MoveL Offs(p0,833.4,751.2, 0), v100, z5, tool0;
	MoveL Offs(p0,832.8656000000001,748.9728, 0), v100, z5, tool0;
	MoveL Offs(p0,832.525,747.825, 0), v100, z5, tool0;
	MoveL Offs(p0,832.1184,746.4911999999999, 0), v100, z5, tool0;
	MoveL Offs(p0,831.6542,744.9966000000001, 0), v100, z5, tool0;
	MoveL Offs(p0,831.1408000000001,743.3664000000001, 0), v100, z5, tool0;
	MoveL Offs(p0,830.5866,741.6258, 0), v100, z5, tool0;
	MoveL Offs(p0,830.0,739.8, 0), v100, z5, tool0;
	MoveL Offs(p0,830.0,739.8, 0), v100, z5, tool0;
	MoveJ Offs(p0,489.0,738.0, 10), v100, z1, tool0;
	MoveL Offs(p0,491.1094000000001,737.3012000000001, 0), v100, z5, tool0;
	MoveL Offs(p0,493.44320000000016,736.5376000000001, 0), v100, z5, tool0;
	MoveL Offs(p0,495.9498,735.7284, 0), v100, z5, tool0;
	MoveL Offs(p0,498.57759999999996,734.8928, 0), v100, z5, tool0;
	MoveL Offs(p0,501.275,734.05, 0), v100, z5, tool0;
	MoveL Offs(p0,503.99039999999997,733.2191999999999, 0), v100, z5, tool0;
	MoveL Offs(p0,506.6722,732.4196, 0), v100, z5, tool0;
	MoveL Offs(p0,509.2688,731.6704000000001, 0), v100, z5, tool0;
	MoveL Offs(p0,511.72860000000003,730.9908, 0), v100, z5, tool0;
	MoveL Offs(p0,514.0,730.4, 0), v100, z5, tool0;
	MoveL Offs(p0,527.0,727.0, 0), v100, z5, tool0;
	MoveL Offs(p0,504.0,726.8, 0), v100, z5, tool0;
	MoveL Offs(p0,499.70680000000004,726.7102000000001, 0), v100, z5, tool0;
	MoveL Offs(p0,495.59840000000014,726.5616000000002, 0), v100, z5, tool0;
	MoveL Offs(p0,491.69159999999994,726.3554, 0), v100, z5, tool0;
	MoveL Offs(p0,488.0032,726.0928, 0), v100, z5, tool0;
	MoveL Offs(p0,484.55,725.775, 0), v100, z5, tool0;
	MoveL Offs(p0,481.3487999999999,725.4032, 0), v100, z5, tool0;
	MoveL Offs(p0,478.41639999999995,724.9786, 0), v100, z5, tool0;
	MoveL Offs(p0,475.76959999999997,724.5024000000001, 0), v100, z5, tool0;
	MoveL Offs(p0,473.4252,723.9757999999999, 0), v100, z5, tool0;
	MoveL Offs(p0,471.4,723.4, 0), v100, z5, tool0;
	MoveL Offs(p0,462.0,720.4, 0), v100, z5, tool0;
	MoveL Offs(p0,454.0,729.6, 0), v100, z5, tool0;
	MoveL Offs(p0,450.84319999999997,733.3776000000001, 0), v100, z5, tool0;
	MoveL Offs(p0,448.4736000000001,736.4688000000002, 0), v100, z5, tool0;
	MoveL Offs(p0,446.92240000000004,738.9312, 0), v100, z5, tool0;
	MoveL Offs(p0,446.22080000000005,740.8224, 0), v100, z5, tool0;
	MoveL Offs(p0,446.4,742.2, 0), v100, z5, tool0;
	MoveL Offs(p0,447.49120000000005,743.1216, 0), v100, z5, tool0;
	MoveL Offs(p0,449.52560000000005,743.6448, 0), v100, z5, tool0;
	MoveL Offs(p0,452.5344000000001,743.8272000000001, 0), v100, z5, tool0;
	MoveL Offs(p0,456.5488,743.7264, 0), v100, z5, tool0;
	MoveL Offs(p0,461.6,743.4, 0), v100, z5, tool0;
	MoveL Offs(p0,464.2302000000001,743.1678, 0), v100, z5, tool0;
	MoveL Offs(p0,467.04160000000013,742.8384000000002, 0), v100, z5, tool0;
	MoveL Offs(p0,469.9753999999999,742.4225999999999, 0), v100, z5, tool0;
	MoveL Offs(p0,472.9728,741.9312, 0), v100, z5, tool0;
	MoveL Offs(p0,475.975,741.375, 0), v100, z5, tool0;
	MoveL Offs(p0,478.9232,740.7648, 0), v100, z5, tool0;
	MoveL Offs(p0,481.7586,740.1114, 0), v100, z5, tool0;
	MoveL Offs(p0,484.42240000000004,739.4256000000001, 0), v100, z5, tool0;
	MoveL Offs(p0,486.8558,738.7182, 0), v100, z5, tool0;
	MoveL Offs(p0,489.0,738.0, 0), v100, z5, tool0;
	MoveL Offs(p0,489.0,738.0, 0), v100, z5, tool0;
	MoveJ Offs(p0,574.2,726.6, 10), v100, z1, tool0;
	MoveL Offs(p0,572.6934,724.2924, 0), v100, z5, tool0;
	MoveL Offs(p0,572.0368000000001,723.3488, 0), v100, z5, tool0;
	MoveL Offs(p0,571.325,722.35, 0), v100, z5, tool0;
	MoveL Offs(p0,570.5712000000001,721.3152000000001, 0), v100, z5, tool0;
	MoveL Offs(p0,569.7886,720.2636, 0), v100, z5, tool0;
	MoveL Offs(p0,568.9904,719.2144000000001, 0), v100, z5, tool0;
	MoveL Offs(p0,568.1898,718.1868000000001, 0), v100, z5, tool0;
	MoveL Offs(p0,567.4,717.2, 0), v100, z5, tool0;
	MoveL Offs(p0,562.8,711.4, 0), v100, z5, tool0;
	MoveL Offs(p0,555.8,715.2, 0), v100, z5, tool0;
	MoveL Offs(p0,553.1776000000002,716.6000000000001, 0), v100, z5, tool0;
	MoveL Offs(p0,551.6564000000001,717.3419999999999, 0), v100, z5, tool0;
	MoveL Offs(p0,550.0368000000001,718.0960000000001, 0), v100, z5, tool0;
	MoveL Offs(p0,548.35,718.85, 0), v100, z5, tool0;
	MoveL Offs(p0,546.6272,719.592, 0), v100, z5, tool0;
	MoveL Offs(p0,544.8996,720.3100000000001, 0), v100, z5, tool0;
	MoveL Offs(p0,543.1984,720.992, 0), v100, z5, tool0;
	MoveL Offs(p0,541.5548000000001,721.626, 0), v100, z5, tool0;
	MoveL Offs(p0,540.0,722.2, 0), v100, z5, tool0;
	MoveL Offs(p0,531.0,725.4, 0), v100, z5, tool0;
	MoveL Offs(p0,544.0,724.6, 0), v100, z5, tool0;
	MoveL Offs(p0,547.2176000000002,724.4162, 0), v100, z5, tool0;
	MoveL Offs(p0,550.2048000000002,724.3536000000001, 0), v100, z5, tool0;
	MoveL Offs(p0,553.0432000000001,724.4254, 0), v100, z5, tool0;
	MoveL Offs(p0,555.8144,724.6448, 0), v100, z5, tool0;
	MoveL Offs(p0,558.6,725.025, 0), v100, z5, tool0;
	MoveL Offs(p0,561.4816000000001,725.5791999999999, 0), v100, z5, tool0;
	MoveL Offs(p0,564.5408,726.3206, 0), v100, z5, tool0;
	MoveL Offs(p0,567.8592000000001,727.2624000000001, 0), v100, z5, tool0;
	MoveL Offs(p0,571.5184,728.4178, 0), v100, z5, tool0;
	MoveL Offs(p0,575.6,729.8, 0), v100, z5, tool0;
	MoveL Offs(p0,574.7488000000001,727.6432000000001, 0), v100, z5, tool0;
	MoveL Offs(p0,574.4876,727.1324000000001, 0), v100, z5, tool0;
	MoveL Offs(p0,574.2,726.6, 0), v100, z5, tool0;
	MoveL Offs(p0,574.2,726.6, 0), v100, z5, tool0;
	MoveJ Offs(p0,372.0,712.4, 10), v100, z1, tool0;
	MoveL Offs(p0,371.20619999999997,709.9988000000001, 0), v100, z5, tool0;
	MoveL Offs(p0,370.6304,708.8416000000001, 0), v100, z5, tool0;
	MoveL Offs(p0,369.925,707.55, 0), v100, z5, tool0;
	MoveL Offs(p0,369.1056,706.1504, 0), v100, z5, tool0;
	MoveL Offs(p0,368.1878,704.6691999999999, 0), v100, z5, tool0;
	MoveL Offs(p0,367.1872,703.1328000000001, 0), v100, z5, tool0;
	MoveL Offs(p0,366.11940000000004,701.5676000000001, 0), v100, z5, tool0;
	MoveL Offs(p0,365.0,700.0, 0), v100, z5, tool0;
	MoveL Offs(p0,360.6804000000001,693.8102000000001, 0), v100, z5, tool0;
	MoveL Offs(p0,356.81920000000014,687.5376000000002, 0), v100, z5, tool0;
	MoveL Offs(p0,353.3827999999999,681.0874, 0), v100, z5, tool0;
	MoveL Offs(p0,350.3376,674.3648000000001, 0), v100, z5, tool0;
	MoveL Offs(p0,347.65,667.275, 0), v100, z5, tool0;
	MoveL Offs(p0,345.2864,659.7232, 0), v100, z5, tool0;
	MoveL Offs(p0,343.2132,651.6146, 0), v100, z5, tool0;
	MoveL Offs(p0,341.39680000000004,642.8543999999999, 0), v100, z5, tool0;
	MoveL Offs(p0,339.8036,633.3478000000001, 0), v100, z5, tool0;
	MoveL Offs(p0,338.4,623.0, 0), v100, z5, tool0;
	MoveL Offs(p0,337.0,611.0, 0), v100, z5, tool0;
	MoveL Offs(p0,319.6,610.4, 0), v100, z5, tool0;
	MoveL Offs(p0,314.14520000000005,610.2422000000001, 0), v100, z5, tool0;
	MoveL Offs(p0,309.82560000000007,610.2176000000002, 0), v100, z5, tool0;
	MoveL Offs(p0,306.52840000000003,610.4594, 0), v100, z5, tool0;
	MoveL Offs(p0,304.1408,611.1008, 0), v100, z5, tool0;
	MoveL Offs(p0,302.55,612.275, 0), v100, z5, tool0;
	MoveL Offs(p0,301.64320000000004,614.1152, 0), v100, z5, tool0;
	MoveL Offs(p0,301.3076,616.7546, 0), v100, z5, tool0;
	MoveL Offs(p0,301.4304,620.3264000000001, 0), v100, z5, tool0;
	MoveL Offs(p0,301.89880000000005,624.9638, 0), v100, z5, tool0;
	MoveL Offs(p0,302.6,630.8, 0), v100, z5, tool0;
	MoveL Offs(p0,304.40600000000006,641.6114, 0), v100, z5, tool0;
	MoveL Offs(p0,307.2560000000001,652.2512000000002, 0), v100, z5, tool0;
	MoveL Offs(p0,311.078,662.6078, 0), v100, z5, tool0;
	MoveL Offs(p0,315.80000000000007,672.5696, 0), v100, z5, tool0;
	MoveL Offs(p0,321.35,682.025, 0), v100, z5, tool0;
	MoveL Offs(p0,327.65600000000006,690.8624, 0), v100, z5, tool0;
	MoveL Offs(p0,334.646,698.9702, 0), v100, z5, tool0;
	MoveL Offs(p0,342.24800000000005,706.2368, 0), v100, z5, tool0;
	MoveL Offs(p0,350.39,712.5506, 0), v100, z5, tool0;
	MoveL Offs(p0,359.0,717.8, 0), v100, z5, tool0;
	MoveL Offs(p0,361.03020000000004,718.8808000000001, 0), v100, z5, tool0;
	MoveL Offs(p0,362.7136000000001,719.7264000000002, 0), v100, z5, tool0;
	MoveL Offs(p0,364.09939999999995,720.3416, 0), v100, z5, tool0;
	MoveL Offs(p0,365.2368,720.7312, 0), v100, z5, tool0;
	MoveL Offs(p0,366.175,720.9, 0), v100, z5, tool0;
	MoveL Offs(p0,366.9632,720.8528, 0), v100, z5, tool0;
	MoveL Offs(p0,367.65060000000005,720.5944, 0), v100, z5, tool0;
	MoveL Offs(p0,368.28640000000007,720.1296, 0), v100, z5, tool0;
	MoveL Offs(p0,368.9198,719.4632, 0), v100, z5, tool0;
	MoveL Offs(p0,369.6,718.6, 0), v100, z5, tool0;
	MoveL Offs(p0,370.96320000000003,716.1007999999999, 0), v100, z5, tool0;
	MoveL Offs(p0,371.25,715.425, 0), v100, z5, tool0;
	MoveL Offs(p0,371.50079999999997,714.7552, 0), v100, z5, tool0;
	MoveL Offs(p0,371.7084,714.1046, 0), v100, z5, tool0;
	MoveL Offs(p0,371.86560000000003,713.4864, 0), v100, z5, tool0;
	MoveL Offs(p0,371.96520000000004,712.9138, 0), v100, z5, tool0;
	MoveL Offs(p0,372.0,712.4, 0), v100, z5, tool0;
	MoveL Offs(p0,372.0,712.4, 0), v100, z5, tool0;
	MoveJ Offs(p0,540.0,716.2, 10), v100, z1, tool0;
	MoveL Offs(p0,542.4624000000001,715.2832000000002, 0), v100, z5, tool0;
	MoveL Offs(p0,543.7926,714.6987999999999, 0), v100, z5, tool0;
	MoveL Offs(p0,545.1551999999999,714.0496, 0), v100, z5, tool0;
	MoveL Offs(p0,546.525,713.35, 0), v100, z5, tool0;
	MoveL Offs(p0,547.8768,712.6144, 0), v100, z5, tool0;
	MoveL Offs(p0,549.1854,711.8572, 0), v100, z5, tool0;
	MoveL Offs(p0,550.4256,711.0928000000001, 0), v100, z5, tool0;
	MoveL Offs(p0,551.5722000000001,710.3356, 0), v100, z5, tool0;
	MoveL Offs(p0,552.6,709.6, 0), v100, z5, tool0;
	MoveL Offs(p0,558.0,705.0, 0), v100, z5, tool0;
	MoveL Offs(p0,544.2,687.2, 0), v100, z5, tool0;
	MoveL Offs(p0,541.9336000000001,684.2560000000001, 0), v100, z5, tool0;
	MoveL Offs(p0,539.6048000000002,681.3360000000002, 0), v100, z5, tool0;
	MoveL Offs(p0,537.2591999999999,678.488, 0), v100, z5, tool0;
	MoveL Offs(p0,534.9424,675.76, 0), v100, z5, tool0;
	MoveL Offs(p0,532.7,673.2, 0), v100, z5, tool0;
	MoveL Offs(p0,530.5776,670.856, 0), v100, z5, tool0;
	MoveL Offs(p0,528.6207999999999,668.776, 0), v100, z5, tool0;
	MoveL Offs(p0,526.8752000000001,667.008, 0), v100, z5, tool0;
	MoveL Offs(p0,525.3864000000001,665.6, 0), v100, z5, tool0;
	MoveL Offs(p0,524.2,664.6, 0), v100, z5, tool0;
	MoveL Offs(p0,521.2336000000001,662.3568000000002, 0), v100, z5, tool0;
	MoveL Offs(p0,520.0654000000001,661.6102, 0), v100, z5, tool0;
	MoveL Offs(p0,519.0448,661.1024, 0), v100, z5, tool0;
	MoveL Offs(p0,518.125,660.825, 0), v100, z5, tool0;
	MoveL Offs(p0,517.2592,660.7696, 0), v100, z5, tool0;
	MoveL Offs(p0,516.4005999999999,660.9278, 0), v100, z5, tool0;
	MoveL Offs(p0,515.5024000000001,661.2912, 0), v100, z5, tool0;
	MoveL Offs(p0,514.5178,661.8514, 0), v100, z5, tool0;
	MoveL Offs(p0,513.4,662.6, 0), v100, z5, tool0;
	MoveL Offs(p0,510.65020000000004,664.8854000000001, 0), v100, z5, tool0;
	MoveL Offs(p0,506.40160000000014,669.0272000000002, 0), v100, z5, tool0;
	MoveL Offs(p0,501.0754,674.5537999999999, 0), v100, z5, tool0;
	MoveL Offs(p0,495.0928,680.9936, 0), v100, z5, tool0;
	MoveL Offs(p0,488.875,687.875, 0), v100, z5, tool0;
	MoveL Offs(p0,482.84319999999997,694.7264, 0), v100, z5, tool0;
	MoveL Offs(p0,477.41859999999997,701.0762000000001, 0), v100, z5, tool0;
	MoveL Offs(p0,473.0224,706.4528, 0), v100, z5, tool0;
	MoveL Offs(p0,470.07579999999996,710.3846000000001, 0), v100, z5, tool0;
	MoveL Offs(p0,469.0,712.4, 0), v100, z5, tool0;
	MoveL Offs(p0,471.625,714.9, 0), v100, z5, tool0;
	MoveL Offs(p0,472.6719999999999,715.4384, 0), v100, z5, tool0;
	MoveL Offs(p0,473.851,715.9672, 0), v100, z5, tool0;
	MoveL Offs(p0,475.14400000000006,716.4768, 0), v100, z5, tool0;
	MoveL Offs(p0,476.533,716.9576, 0), v100, z5, tool0;
	MoveL Offs(p0,478.0,717.4, 0), v100, z5, tool0;
	MoveL Offs(p0,482.0796,718.1386000000001, 0), v100, z5, tool0;
	MoveL Offs(p0,487.5968000000001,718.6768000000002, 0), v100, z5, tool0;
	MoveL Offs(p0,494.18919999999997,719.0181999999999, 0), v100, z5, tool0;
	MoveL Offs(p0,501.49440000000016,719.1664000000001, 0), v100, z5, tool0;
	MoveL Offs(p0,509.15,719.125, 0), v100, z5, tool0;
	MoveL Offs(p0,516.7936,718.8976, 0), v100, z5, tool0;
	MoveL Offs(p0,524.0628,718.4878000000001, 0), v100, z5, tool0;
	MoveL Offs(p0,530.5952,717.8992000000001, 0), v100, z5, tool0;
	MoveL Offs(p0,536.0283999999999,717.1354, 0), v100, z5, tool0;
	MoveL Offs(p0,540.0,716.2, 0), v100, z5, tool0;
	MoveL Offs(p0,540.0,716.2, 0), v100, z5, tool0;
	MoveJ Offs(p0,668.4,709.0, 10), v100, z1, tool0;
	MoveL Offs(p0,668.5120000000001,706.1360000000002, 0), v100, z5, tool0;
	MoveL Offs(p0,668.292,704.9860000000001, 0), v100, z5, tool0;
	MoveL Offs(p0,667.8080000000001,703.9440000000002, 0), v100, z5, tool0;
	MoveL Offs(p0,667.0,702.95, 0), v100, z5, tool0;
	MoveL Offs(p0,665.808,701.9440000000001, 0), v100, z5, tool0;
	MoveL Offs(p0,664.1719999999999,700.866, 0), v100, z5, tool0;
	MoveL Offs(p0,662.0319999999999,699.6560000000001, 0), v100, z5, tool0;
	MoveL Offs(p0,659.3280000000001,698.2540000000001, 0), v100, z5, tool0;
	MoveL Offs(p0,656.0,696.6, 0), v100, z5, tool0;
	MoveL Offs(p0,650.2782,693.907, 0), v100, z5, tool0;
	MoveL Offs(p0,644.7616,691.4720000000003, 0), v100, z5, tool0;
	MoveL Offs(p0,639.4633999999999,689.301, 0), v100, z5, tool0;
	MoveL Offs(p0,634.3968000000001,687.4000000000001, 0), v100, z5, tool0;
	MoveL Offs(p0,629.575,685.775, 0), v100, z5, tool0;
	MoveL Offs(p0,625.0112,684.432, 0), v100, z5, tool0;
	MoveL Offs(p0,620.7185999999999,683.3770000000001, 0), v100, z5, tool0;
	MoveL Offs(p0,616.7104000000002,682.6160000000001, 0), v100, z5, tool0;
	MoveL Offs(p0,612.9998,682.155, 0), v100, z5, tool0;
	MoveL Offs(p0,609.6,682.0, 0), v100, z5, tool0;
	MoveL Offs(p0,606.7790000000002,682.0202, 0), v100, z5, tool0;
	MoveL Offs(p0,604.5280000000001,682.1136000000002, 0), v100, z5, tool0;
	MoveL Offs(p0,602.8050000000001,682.3293999999999, 0), v100, z5, tool0;
	MoveL Offs(p0,601.568,682.7168, 0), v100, z5, tool0;
	MoveL Offs(p0,600.775,683.325, 0), v100, z5, tool0;
	MoveL Offs(p0,600.3839999999999,684.2031999999999, 0), v100, z5, tool0;
	MoveL Offs(p0,600.3530000000001,685.4005999999999, 0), v100, z5, tool0;
	MoveL Offs(p0,600.6400000000001,686.9664, 0), v100, z5, tool0;
	MoveL Offs(p0,601.2030000000001,688.9498, 0), v100, z5, tool0;
	MoveL Offs(p0,602.0,691.4, 0), v100, z5, tool0;
	MoveL Offs(p0,603.2432000000001,694.0432000000002, 0), v100, z5, tool0;
	MoveL Offs(p0,604.0898,695.1548, 0), v100, z5, tool0;
	MoveL Offs(p0,605.1776000000001,696.1776000000001, 0), v100, z5, tool0;
	MoveL Offs(p0,606.575,697.15, 0), v100, z5, tool0;
	MoveL Offs(p0,608.3504,698.1104, 0), v100, z5, tool0;
	MoveL Offs(p0,610.5722,699.0971999999999, 0), v100, z5, tool0;
	MoveL Offs(p0,613.3088,700.1488000000002, 0), v100, z5, tool0;
	MoveL Offs(p0,616.6286,701.3036, 0), v100, z5, tool0;
	MoveL Offs(p0,620.6,702.6, 0), v100, z5, tool0;
	MoveL Offs(p0,623.4330000000001,703.5560000000002, 0), v100, z5, tool0;
	MoveL Offs(p0,626.488,704.6080000000002, 0), v100, z5, tool0;
	MoveL Offs(p0,629.699,705.732, 0), v100, z5, tool0;
	MoveL Offs(p0,633.0000000000001,706.904, 0), v100, z5, tool0;
	MoveL Offs(p0,636.325,708.1, 0), v100, z5, tool0;
	MoveL Offs(p0,639.608,709.296, 0), v100, z5, tool0;
	MoveL Offs(p0,642.783,710.4680000000001, 0), v100, z5, tool0;
	MoveL Offs(p0,645.784,711.5920000000001, 0), v100, z5, tool0;
	MoveL Offs(p0,648.5450000000001,712.644, 0), v100, z5, tool0;
	MoveL Offs(p0,651.0,713.6, 0), v100, z5, tool0;
	MoveL Offs(p0,655.0998000000002,715.2100000000002, 0), v100, z5, tool0;
	MoveL Offs(p0,658.4544000000002,716.4240000000002, 0), v100, z5, tool0;
	MoveL Offs(p0,661.1465999999999,717.218, 0), v100, z5, tool0;
	MoveL Offs(p0,663.2592000000001,717.5680000000001, 0), v100, z5, tool0;
	MoveL Offs(p0,664.875,717.45, 0), v100, z5, tool0;
	MoveL Offs(p0,666.0768,716.8399999999999, 0), v100, z5, tool0;
	MoveL Offs(p0,666.9474,715.714, 0), v100, z5, tool0;
	MoveL Offs(p0,667.5696,714.048, 0), v100, z5, tool0;
	MoveL Offs(p0,668.0262,711.818, 0), v100, z5, tool0;
	MoveL Offs(p0,668.4,709.0, 0), v100, z5, tool0;
	MoveL Offs(p0,668.4,709.0, 0), v100, z5, tool0;
	MoveJ Offs(p0,398.8,700.8, 10), v100, z1, tool0;
	MoveL Offs(p0,403.3928000000001,698.0432000000001, 0), v100, z5, tool0;
	MoveL Offs(p0,407.0064000000001,695.8096000000003, 0), v100, z5, tool0;
	MoveL Offs(p0,409.69360000000006,693.9744, 0), v100, z5, tool0;
	MoveL Offs(p0,411.5072000000001,692.4128, 0), v100, z5, tool0;
	MoveL Offs(p0,412.5,691.0, 0), v100, z5, tool0;
	MoveL Offs(p0,412.7248000000001,689.6112, 0), v100, z5, tool0;
	MoveL Offs(p0,412.2344,688.1216000000001, 0), v100, z5, tool0;
	MoveL Offs(p0,411.0816000000001,686.4064000000001, 0), v100, z5, tool0;
	MoveL Offs(p0,409.3192,684.3408000000002, 0), v100, z5, tool0;
	MoveL Offs(p0,407.0,681.8, 0), v100, z5, tool0;
	MoveL Offs(p0,403.25300000000004,677.2300000000001, 0), v100, z5, tool0;
	MoveL Offs(p0,399.8240000000001,672.1920000000001, 0), v100, z5, tool0;
	MoveL Offs(p0,396.731,666.7339999999999, 0), v100, z5, tool0;
	MoveL Offs(p0,393.992,660.904, 0), v100, z5, tool0;
	MoveL Offs(p0,391.625,654.75, 0), v100, z5, tool0;
	MoveL Offs(p0,389.64799999999997,648.3199999999999, 0), v100, z5, tool0;
	MoveL Offs(p0,388.079,641.662, 0), v100, z5, tool0;
	MoveL Offs(p0,386.93600000000004,634.824, 0), v100, z5, tool0;
	MoveL Offs(p0,386.237,627.854, 0), v100, z5, tool0;
	MoveL Offs(p0,386.0,620.8, 0), v100, z5, tool0;
	MoveL Offs(p0,386.0,612.6, 0), v100, z5, tool0;
	MoveL Offs(p0,373.8,611.2, 0), v100, z5, tool0;
	MoveL Offs(p0,369.36920000000003,610.8163999999999, 0), v100, z5, tool0;
	MoveL Offs(p0,365.01760000000013,610.5072000000002, 0), v100, z5, tool0;
	MoveL Offs(p0,360.83639999999997,610.2748, 0), v100, z5, tool0;
	MoveL Offs(p0,356.9168,610.1216000000001, 0), v100, z5, tool0;
	MoveL Offs(p0,353.35,610.05, 0), v100, z5, tool0;
	MoveL Offs(p0,350.2272,610.0624, 0), v100, z5, tool0;
	MoveL Offs(p0,347.6396,610.1612, 0), v100, z5, tool0;
	MoveL Offs(p0,345.67840000000007,610.3488, 0), v100, z5, tool0;
	MoveL Offs(p0,344.4348,610.6276, 0), v100, z5, tool0;
	MoveL Offs(p0,344.0,611.0, 0), v100, z5, tool0;
	MoveL Offs(p0,344.1936,613.9570000000001, 0), v100, z5, tool0;
	MoveL Offs(p0,344.7328000000001,618.2880000000002, 0), v100, z5, tool0;
	MoveL Offs(p0,345.55519999999996,623.6630000000001, 0), v100, z5, tool0;
	MoveL Offs(p0,346.59839999999997,629.7520000000001, 0), v100, z5, tool0;
	MoveL Offs(p0,347.8,636.225, 0), v100, z5, tool0;
	MoveL Offs(p0,349.09759999999994,642.7520000000001, 0), v100, z5, tool0;
	MoveL Offs(p0,350.4288,649.0029999999999, 0), v100, z5, tool0;
	MoveL Offs(p0,351.73120000000006,654.6480000000001, 0), v100, z5, tool0;
	MoveL Offs(p0,352.9424,659.3570000000001, 0), v100, z5, tool0;
	MoveL Offs(p0,354.0,662.8, 0), v100, z5, tool0;
	MoveL Offs(p0,355.3784,666.5536, 0), v100, z5, tool0;
	MoveL Offs(p0,356.9632000000001,670.4368000000002, 0), v100, z5, tool0;
	MoveL Offs(p0,358.7088,674.3632, 0), v100, z5, tool0;
	MoveL Offs(p0,360.56960000000004,678.2464, 0), v100, z5, tool0;
	MoveL Offs(p0,362.5,682.0, 0), v100, z5, tool0;
	MoveL Offs(p0,364.4544,685.5375999999999, 0), v100, z5, tool0;
	MoveL Offs(p0,366.3872,688.7728, 0), v100, z5, tool0;
	MoveL Offs(p0,368.25280000000004,691.6192000000001, 0), v100, z5, tool0;
	MoveL Offs(p0,370.0056,693.9904, 0), v100, z5, tool0;
	MoveL Offs(p0,371.6,695.8, 0), v100, z5, tool0;
	MoveL Offs(p0,373.78560000000004,698.4176, 0), v100, z5, tool0;
	MoveL Offs(p0,374.425,699.225, 0), v100, z5, tool0;
	MoveL Offs(p0,375.07039999999995,700.0624, 0), v100, z5, tool0;
	MoveL Offs(p0,375.70619999999997,700.9141999999999, 0), v100, z5, tool0;
	MoveL Offs(p0,376.31680000000006,701.7648000000002, 0), v100, z5, tool0;
	MoveL Offs(p0,376.88660000000004,702.5986, 0), v100, z5, tool0;
	MoveL Offs(p0,377.4,703.4, 0), v100, z5, tool0;
	MoveL Offs(p0,379.8560000000001,706.1056000000002, 0), v100, z5, tool0;
	MoveL Offs(p0,381.27899999999994,706.8704, 0), v100, z5, tool0;
	MoveL Offs(p0,382.88800000000003,707.2367999999999, 0), v100, z5, tool0;
	MoveL Offs(p0,384.725,707.2, 0), v100, z5, tool0;
	MoveL Offs(p0,386.832,706.7552, 0), v100, z5, tool0;
	MoveL Offs(p0,389.25100000000003,705.8976, 0), v100, z5, tool0;
	MoveL Offs(p0,392.024,704.6224, 0), v100, z5, tool0;
	MoveL Offs(p0,395.19300000000004,702.9248, 0), v100, z5, tool0;
	MoveL Offs(p0,398.8,700.8, 0), v100, z5, tool0;
	MoveL Offs(p0,398.8,700.8, 0), v100, z5, tool0;
	MoveJ Offs(p0,696.8,701.6, 10), v100, z1, tool0;
	MoveL Offs(p0,698.285,699.1915999999999, 0), v100, z5, tool0;
	MoveL Offs(p0,698.704,698.3232, 0), v100, z5, tool0;
	MoveL Offs(p0,699.075,697.45, 0), v100, z5, tool0;
	MoveL Offs(p0,699.392,696.5888000000001, 0), v100, z5, tool0;
	MoveL Offs(p0,699.649,695.7564, 0), v100, z5, tool0;
	MoveL Offs(p0,699.84,694.9696000000001, 0), v100, z5, tool0;
	MoveL Offs(p0,699.9590000000001,694.2452000000001, 0), v100, z5, tool0;
	MoveL Offs(p0,700.0,693.6, 0), v100, z5, tool0;
	MoveL Offs(p0,699.1600000000002,691.2064000000001, 0), v100, z5, tool0;
	MoveL Offs(p0,698.164,689.2026, 0), v100, z5, tool0;
	MoveL Offs(p0,696.8320000000001,686.7392000000001, 0), v100, z5, tool0;
	MoveL Offs(p0,695.2,683.875, 0), v100, z5, tool0;
	MoveL Offs(p0,693.304,680.6687999999999, 0), v100, z5, tool0;
	MoveL Offs(p0,691.18,677.1794, 0), v100, z5, tool0;
	MoveL Offs(p0,688.8640000000001,673.4656000000001, 0), v100, z5, tool0;
	MoveL Offs(p0,686.392,669.5862, 0), v100, z5, tool0;
	MoveL Offs(p0,683.8,665.6, 0), v100, z5, tool0;
	MoveL Offs(p0,678.2588000000002,657.1580000000001, 0), v100, z5, tool0;
	MoveL Offs(p0,673.3824000000002,649.4480000000001, 0), v100, z5, tool0;
	MoveL Offs(p0,669.1515999999999,642.434, 0), v100, z5, tool0;
	MoveL Offs(p0,665.5472000000002,636.08, 0), v100, z5, tool0;
	MoveL Offs(p0,662.55,630.35, 0), v100, z5, tool0;
	MoveL Offs(p0,660.1408,625.208, 0), v100, z5, tool0;
	MoveL Offs(p0,658.3003999999999,620.6179999999999, 0), v100, z5, tool0;
	MoveL Offs(p0,657.0096000000001,616.5440000000001, 0), v100, z5, tool0;
	MoveL Offs(p0,656.2492,612.95, 0), v100, z5, tool0;
	MoveL Offs(p0,656.0,609.8, 0), v100, z5, tool0;
	MoveL Offs(p0,656.2054,606.5512000000001, 0), v100, z5, tool0;
	MoveL Offs(p0,656.7792000000002,602.6976000000002, 0), v100, z5, tool0;
	MoveL Offs(p0,657.6578,598.4384, 0), v100, z5, tool0;
	MoveL Offs(p0,658.7776000000001,593.9728, 0), v100, z5, tool0;
	MoveL Offs(p0,660.075,589.5, 0), v100, z5, tool0;
	MoveL Offs(p0,661.4864,585.2191999999999, 0), v100, z5, tool0;
	MoveL Offs(p0,662.9482,581.3296, 0), v100, z5, tool0;
	MoveL Offs(p0,664.3968000000001,578.0304, 0), v100, z5, tool0;
	MoveL Offs(p0,665.7686,575.5208, 0), v100, z5, tool0;
	MoveL Offs(p0,667.0,574.0, 0), v100, z5, tool0;
	MoveL Offs(p0,669.6351999999999,572.7724000000001, 0), v100, z5, tool0;
	MoveL Offs(p0,670.8943999999999,572.3968000000002, 0), v100, z5, tool0;
	MoveL Offs(p0,672.3,572.05, 0), v100, z5, tool0;
	MoveL Offs(p0,673.8256,571.7392, 0), v100, z5, tool0;
	MoveL Offs(p0,675.4448,571.4716000000001, 0), v100, z5, tool0;
	MoveL Offs(p0,677.1312,571.2544, 0), v100, z5, tool0;
	MoveL Offs(p0,678.8584,571.0948000000001, 0), v100, z5, tool0;
	MoveL Offs(p0,680.6,571.0, 0), v100, z5, tool0;
	MoveL Offs(p0,683.0916,570.8158000000001, 0), v100, z5, tool0;
	MoveL Offs(p0,685.1968000000003,570.6064000000001, 0), v100, z5, tool0;
	MoveL Offs(p0,686.9612,570.3466000000001, 0), v100, z5, tool0;
	MoveL Offs(p0,688.4304000000001,570.0112000000001, 0), v100, z5, tool0;
	MoveL Offs(p0,689.65,569.575, 0), v100, z5, tool0;
	MoveL Offs(p0,690.6656,569.0128, 0), v100, z5, tool0;
	MoveL Offs(p0,691.5228,568.2994000000001, 0), v100, z5, tool0;
	MoveL Offs(p0,692.2672,567.4096000000001, 0), v100, z5, tool0;
	MoveL Offs(p0,692.9444000000001,566.3181999999999, 0), v100, z5, tool0;
	MoveL Offs(p0,693.6,565.0, 0), v100, z5, tool0;
	MoveL Offs(p0,695.0592000000001,561.0704000000002, 0), v100, z5, tool0;
	MoveL Offs(p0,695.3477999999999,559.1086, 0), v100, z5, tool0;
	MoveL Offs(p0,695.3376000000001,557.1312, 0), v100, z5, tool0;
	MoveL Offs(p0,695.025,555.125, 0), v100, z5, tool0;
	MoveL Offs(p0,694.4064000000001,553.0768, 0), v100, z5, tool0;
	MoveL Offs(p0,693.4782,550.9734000000001, 0), v100, z5, tool0;
	MoveL Offs(p0,692.2368,548.8016, 0), v100, z5, tool0;
	MoveL Offs(p0,690.6786,546.5482, 0), v100, z5, tool0;
	MoveL Offs(p0,688.8,544.2, 0), v100, z5, tool0;
	MoveL Offs(p0,686.4798,541.2983999999999, 0), v100, z5, tool0;
	MoveL Offs(p0,685.8176000000001,540.3728, 0), v100, z5, tool0;
	MoveL Offs(p0,685.225,539.5, 0), v100, z5, tool0;
	MoveL Offs(p0,684.7104,538.6991999999999, 0), v100, z5, tool0;
	MoveL Offs(p0,684.2822,537.9896000000001, 0), v100, z5, tool0;
	MoveL Offs(p0,683.9488,537.3904, 0), v100, z5, tool0;
	MoveL Offs(p0,683.7185999999999,536.9208000000001, 0), v100, z5, tool0;
	MoveL Offs(p0,683.6,536.6, 0), v100, z5, tool0;
	MoveL Offs(p0,682.8000000000002,533.8752000000002, 0), v100, z5, tool0;
	MoveL Offs(p0,681.9259999999999,531.8677999999999, 0), v100, z5, tool0;
	MoveL Offs(p0,680.8480000000001,529.6336, 0), v100, z5, tool0;
	MoveL Offs(p0,679.65,527.325, 0), v100, z5, tool0;
	MoveL Offs(p0,678.4159999999999,525.0944000000001, 0), v100, z5, tool0;
	MoveL Offs(p0,677.2299999999999,523.0941999999999, 0), v100, z5, tool0;
	MoveL Offs(p0,676.176,521.4768, 0), v100, z5, tool0;
	MoveL Offs(p0,675.338,520.3946, 0), v100, z5, tool0;
	MoveL Offs(p0,674.8,520.0, 0), v100, z5, tool0;
	MoveL Offs(p0,674.9782,522.187, 0), v100, z5, tool0;
	MoveL Offs(p0,675.2,522.6, 0), v100, z5, tool0;
	MoveL Offs(p0,673.6,520.725, 0), v100, z5, tool0;
	MoveL Offs(p0,673.3728,519.9296, 0), v100, z5, tool0;
	MoveL Offs(p0,673.1744,519.0838, 0), v100, z5, tool0;
	MoveL Offs(p0,673.0096000000001,518.2032000000002, 0), v100, z5, tool0;
	MoveL Offs(p0,672.8832,517.3034, 0), v100, z5, tool0;
	MoveL Offs(p0,672.8,516.4, 0), v100, z5, tool0;
	MoveL Offs(p0,672.4480000000002,513.9568000000002, 0), v100, z5, tool0;
	MoveL Offs(p0,672.197,512.3122000000001, 0), v100, z5, tool0;
	MoveL Offs(p0,671.9040000000001,510.4384, 0), v100, z5, tool0;
	MoveL Offs(p0,671.575,508.375, 0), v100, z5, tool0;
	MoveL Offs(p0,671.216,506.1616, 0), v100, z5, tool0;
	MoveL Offs(p0,670.833,503.83779999999996, 0), v100, z5, tool0;
	MoveL Offs(p0,670.432,501.44320000000005, 0), v100, z5, tool0;
	MoveL Offs(p0,670.019,499.0174, 0), v100, z5, tool0;
	MoveL Offs(p0,669.6,496.6, 0), v100, z5, tool0;
	MoveL Offs(p0,667.0,482.4, 0), v100, z5, tool0;
	MoveL Offs(p0,656.0,503.4, 0), v100, z5, tool0;
	MoveL Offs(p0,650.2952000000001,514.1646000000001, 0), v100, z5, tool0;
	MoveL Offs(p0,644.8496000000001,524.2128000000001, 0), v100, z5, tool0;
	MoveL Offs(p0,639.7063999999998,533.4762000000001, 0), v100, z5, tool0;
	MoveL Offs(p0,634.9088,541.8864000000001, 0), v100, z5, tool0;
	MoveL Offs(p0,630.5,549.375, 0), v100, z5, tool0;
	MoveL Offs(p0,626.5232,555.8736000000001, 0), v100, z5, tool0;
	MoveL Offs(p0,623.0215999999999,561.3138, 0), v100, z5, tool0;
	MoveL Offs(p0,620.0384,565.6272000000001, 0), v100, z5, tool0;
	MoveL Offs(p0,617.6168,568.7454, 0), v100, z5, tool0;
	MoveL Offs(p0,615.8,570.6, 0), v100, z5, tool0;
	MoveL Offs(p0,613.6236000000001,571.9016, 0), v100, z5, tool0;
	MoveL Offs(p0,611.1088000000002,572.9248000000001, 0), v100, z5, tool0;
	MoveL Offs(p0,608.3372,573.6672, 0), v100, z5, tool0;
	MoveL Offs(p0,605.3904,574.1264, 0), v100, z5, tool0;
	MoveL Offs(p0,602.35,574.3, 0), v100, z5, tool0;
	MoveL Offs(p0,599.2976000000001,574.1856, 0), v100, z5, tool0;
	MoveL Offs(p0,596.3147999999999,573.7808000000001, 0), v100, z5, tool0;
	MoveL Offs(p0,593.4832,573.0832, 0), v100, z5, tool0;
	MoveL Offs(p0,590.8844,572.0904, 0), v100, z5, tool0;
	MoveL Offs(p0,588.6,570.8, 0), v100, z5, tool0;
	MoveL Offs(p0,585.2944000000001,569.1760000000002, 0), v100, z5, tool0;
	MoveL Offs(p0,583.4736,568.595, 0), v100, z5, tool0;
	MoveL Offs(p0,581.5952,568.176, 0), v100, z5, tool0;
	MoveL Offs(p0,579.7,567.925, 0), v100, z5, tool0;
	MoveL Offs(p0,577.8288,567.848, 0), v100, z5, tool0;
	MoveL Offs(p0,576.0224000000001,567.951, 0), v100, z5, tool0;
	MoveL Offs(p0,574.3216,568.2400000000001, 0), v100, z5, tool0;
	MoveL Offs(p0,572.7672,568.721, 0), v100, z5, tool0;
	MoveL Offs(p0,571.4,569.4, 0), v100, z5, tool0;
	MoveL Offs(p0,572.8112,571.848, 0), v100, z5, tool0;
	MoveL Offs(p0,573.5126,572.4939999999999, 0), v100, z5, tool0;
	MoveL Offs(p0,574.3184000000001,573.176, 0), v100, z5, tool0;
	MoveL Offs(p0,575.2178,573.8820000000001, 0), v100, z5, tool0;
	MoveL Offs(p0,576.2,574.6, 0), v100, z5, tool0;
	MoveL Offs(p0,580.4882,578.2042000000001, 0), v100, z5, tool0;
	MoveL Offs(p0,583.9856000000001,582.4816000000001, 0), v100, z5, tool0;
	MoveL Offs(p0,586.6814,587.3494, 0), v100, z5, tool0;
	MoveL Offs(p0,588.5648000000001,592.7248000000001, 0), v100, z5, tool0;
	MoveL Offs(p0,589.625,598.525, 0), v100, z5, tool0;
	MoveL Offs(p0,589.8512,604.6672000000001, 0), v100, z5, tool0;
	MoveL Offs(p0,589.2325999999999,611.0686, 0), v100, z5, tool0;
	MoveL Offs(p0,587.7584,617.6464, 0), v100, z5, tool0;
	MoveL Offs(p0,585.4177999999999,624.3178, 0), v100, z5, tool0;
	MoveL Offs(p0,582.2,631.0, 0), v100, z5, tool0;
	MoveL Offs(p0,576.0,642.6, 0), v100, z5, tool0;
	MoveL Offs(p0,584.2,657.8, 0), v100, z5, tool0;
	MoveL Offs(p0,587.2754000000001,663.4174, 0), v100, z5, tool0;
	MoveL Offs(p0,589.7472000000001,667.8672000000003, 0), v100, z5, tool0;
	MoveL Offs(p0,591.7438000000001,671.2657999999999, 0), v100, z5, tool0;
	MoveL Offs(p0,593.3936,673.7296, 0), v100, z5, tool0;
	MoveL Offs(p0,594.825,675.375, 0), v100, z5, tool0;
	MoveL Offs(p0,596.1664000000001,676.3184, 0), v100, z5, tool0;
	MoveL Offs(p0,597.5462,676.6762000000001, 0), v100, z5, tool0;
	MoveL Offs(p0,599.0928000000001,676.5648, 0), v100, z5, tool0;
	MoveL Offs(p0,600.9346,676.1006000000001, 0), v100, z5, tool0;
	MoveL Offs(p0,603.2,675.4, 0), v100, z5, tool0;
	MoveL Offs(p0,606.2576000000001,674.6560000000002, 0), v100, z5, tool0;
	MoveL Offs(p0,607.7774,674.4460000000001, 0), v100, z5, tool0;
	MoveL Offs(p0,609.3248000000001,674.344, 0), v100, z5, tool0;
	MoveL Offs(p0,610.925,674.35, 0), v100, z5, tool0;
	MoveL Offs(p0,612.6032,674.464, 0), v100, z5, tool0;
	MoveL Offs(p0,614.3846,674.686, 0), v100, z5, tool0;
	MoveL Offs(p0,616.2944,675.016, 0), v100, z5, tool0;
	MoveL Offs(p0,618.3578,675.4540000000001, 0), v100, z5, tool0;
	MoveL Offs(p0,620.6,676.0, 0), v100, z5, tool0;
	MoveL Offs(p0,624.0924000000002,677.0146000000002, 0), v100, z5, tool0;
	MoveL Offs(p0,628.8832000000002,678.6688000000001, 0), v100, z5, tool0;
	MoveL Offs(p0,634.7227999999999,680.8581999999999, 0), v100, z5, tool0;
	MoveL Offs(p0,641.3616,683.4784000000001, 0), v100, z5, tool0;
	MoveL Offs(p0,648.55,686.425, 0), v100, z5, tool0;
	MoveL Offs(p0,656.0384,689.5935999999999, 0), v100, z5, tool0;
	MoveL Offs(p0,663.5772,692.8797999999999, 0), v100, z5, tool0;
	MoveL Offs(p0,670.9168000000001,696.1792, 0), v100, z5, tool0;
	MoveL Offs(p0,677.8076,699.3874000000001, 0), v100, z5, tool0;
	MoveL Offs(p0,684.0,702.4, 0), v100, z5, tool0;
	MoveL Offs(p0,686.4482,703.5872000000002, 0), v100, z5, tool0;
	MoveL Offs(p0,688.4416000000002,704.5056000000002, 0), v100, z5, tool0;
	MoveL Offs(p0,690.0534,705.1504, 0), v100, z5, tool0;
	MoveL Offs(p0,691.3568,705.5168000000001, 0), v100, z5, tool0;
	MoveL Offs(p0,692.425,705.6, 0), v100, z5, tool0;
	MoveL Offs(p0,693.3311999999999,705.3952, 0), v100, z5, tool0;
	MoveL Offs(p0,694.1486000000001,704.8976, 0), v100, z5, tool0;
	MoveL Offs(p0,694.9504000000001,704.1024000000001, 0), v100, z5, tool0;
	MoveL Offs(p0,695.8098,703.0048, 0), v100, z5, tool0;
	MoveL Offs(p0,696.8,701.6, 0), v100, z5, tool0;
	MoveL Offs(p0,696.8,701.6, 0), v100, z5, tool0;
	MoveJ Offs(p0,435.8,657.2, 10), v100, z1, tool0;
	MoveL Offs(p0,437.45820000000015,653.4010000000001, 0), v100, z5, tool0;
	MoveL Offs(p0,439.0576000000002,649.6080000000002, 0), v100, z5, tool0;
	MoveL Offs(p0,440.5753999999999,645.887, 0), v100, z5, tool0;
	MoveL Offs(p0,441.98879999999997,642.3040000000001, 0), v100, z5, tool0;
	MoveL Offs(p0,443.275,638.925, 0), v100, z5, tool0;
	MoveL Offs(p0,444.4112,635.816, 0), v100, z5, tool0;
	MoveL Offs(p0,445.3746,633.043, 0), v100, z5, tool0;
	MoveL Offs(p0,446.1424,630.6720000000001, 0), v100, z5, tool0;
	MoveL Offs(p0,446.69180000000006,628.769, 0), v100, z5, tool0;
	MoveL Offs(p0,447.0,627.4, 0), v100, z5, tool0;
	MoveL Offs(p0,448.4,620.6, 0), v100, z5, tool0;
	MoveL Offs(p0,433.6,618.4, 0), v100, z5, tool0;
	MoveL Offs(p0,431.0774,618.0292000000002, 0), v100, z5, tool0;
	MoveL Offs(p0,428.34720000000016,617.6416000000002, 0), v100, z5, tool0;
	MoveL Offs(p0,425.46579999999994,617.2444, 0), v100, z5, tool0;
	MoveL Offs(p0,422.48960000000005,616.8448, 0), v100, z5, tool0;
	MoveL Offs(p0,419.475,616.45, 0), v100, z5, tool0;
	MoveL Offs(p0,416.47839999999997,616.0672000000001, 0), v100, z5, tool0;
	MoveL Offs(p0,413.5562,615.7036, 0), v100, z5, tool0;
	MoveL Offs(p0,410.76480000000004,615.3664000000001, 0), v100, z5, tool0;
	MoveL Offs(p0,408.1606,615.0628, 0), v100, z5, tool0;
	MoveL Offs(p0,405.8,614.8, 0), v100, z5, tool0;
	MoveL Offs(p0,392.8,613.6, 0), v100, z5, tool0;
	MoveL Offs(p0,393.6,627.2, 0), v100, z5, tool0;
	MoveL Offs(p0,394.10760000000005,633.4778, 0), v100, z5, tool0;
	MoveL Offs(p0,394.9248000000001,639.3824000000002, 0), v100, z5, tool0;
	MoveL Offs(p0,396.07320000000004,644.9605999999999, 0), v100, z5, tool0;
	MoveL Offs(p0,397.5744000000001,650.2592000000001, 0), v100, z5, tool0;
	MoveL Offs(p0,399.45,655.325, 0), v100, z5, tool0;
	MoveL Offs(p0,401.72159999999997,660.2048, 0), v100, z5, tool0;
	MoveL Offs(p0,404.4108,664.9454, 0), v100, z5, tool0;
	MoveL Offs(p0,407.53920000000005,669.5936, 0), v100, z5, tool0;
	MoveL Offs(p0,411.12840000000006,674.1962, 0), v100, z5, tool0;
	MoveL Offs(p0,415.2,678.8, 0), v100, z5, tool0;
	MoveL Offs(p0,417.44540000000006,681.3164, 0), v100, z5, tool0;
	MoveL Offs(p0,419.24320000000006,683.2352000000003, 0), v100, z5, tool0;
	MoveL Offs(p0,420.7458,684.3908, 0), v100, z5, tool0;
	MoveL Offs(p0,422.10560000000004,684.6176000000002, 0), v100, z5, tool0;
	MoveL Offs(p0,423.475,683.75, 0), v100, z5, tool0;
	MoveL Offs(p0,425.00640000000004,681.6224, 0), v100, z5, tool0;
	MoveL Offs(p0,426.8522,678.0691999999999, 0), v100, z5, tool0;
	MoveL Offs(p0,429.1648000000001,672.9248, 0), v100, z5, tool0;
	MoveL Offs(p0,432.0966,666.0236, 0), v100, z5, tool0;
	MoveL Offs(p0,435.8,657.2, 0), v100, z5, tool0;
	MoveL Offs(p0,435.8,657.2, 0), v100, z5, tool0;
	MoveJ Offs(p0,579.6,624.0, 10), v100, z1, tool0;
	MoveL Offs(p0,581.2256,620.0982000000001, 0), v100, z5, tool0;
	MoveL Offs(p0,582.5008000000001,615.8016, 0), v100, z5, tool0;
	MoveL Offs(p0,583.4232,611.2434, 0), v100, z5, tool0;
	MoveL Offs(p0,583.9904,606.5568000000001, 0), v100, z5, tool0;
	MoveL Offs(p0,584.2,601.875, 0), v100, z5, tool0;
	MoveL Offs(p0,584.0495999999999,597.3311999999999, 0), v100, z5, tool0;
	MoveL Offs(p0,583.5368000000001,593.0586, 0), v100, z5, tool0;
	MoveL Offs(p0,582.6592,589.1904000000001, 0), v100, z5, tool0;
	MoveL Offs(p0,581.4144,585.8598, 0), v100, z5, tool0;
	MoveL Offs(p0,579.8,583.2, 0), v100, z5, tool0;
	MoveL Offs(p0,576.9376000000002,580.2304000000001, 0), v100, z5, tool0;
	MoveL Offs(p0,575.5664,579.2256, 0), v100, z5, tool0;
	MoveL Offs(p0,574.2768000000001,578.5472000000001, 0), v100, z5, tool0;
	MoveL Offs(p0,573.1,578.2, 0), v100, z5, tool0;
	MoveL Offs(p0,572.0672000000001,578.1888, 0), v100, z5, tool0;
	MoveL Offs(p0,571.2095999999999,578.5183999999999, 0), v100, z5, tool0;
	MoveL Offs(p0,570.5584000000001,579.1936000000001, 0), v100, z5, tool0;
	MoveL Offs(p0,570.1448,580.2192, 0), v100, z5, tool0;
	MoveL Offs(p0,570.0,581.6, 0), v100, z5, tool0;
	MoveL Offs(p0,569.2493999999999,584.4584, 0), v100, z5, tool0;
	MoveL Offs(p0,568.7008000000001,585.8048000000001, 0), v100, z5, tool0;
	MoveL Offs(p0,568.025,587.3, 0), v100, z5, tool0;
	MoveL Offs(p0,567.2352,588.9152, 0), v100, z5, tool0;
	MoveL Offs(p0,566.3446,590.6216000000001, 0), v100, z5, tool0;
	MoveL Offs(p0,565.3664000000001,592.3904, 0), v100, z5, tool0;
	MoveL Offs(p0,564.3138000000001,594.1928, 0), v100, z5, tool0;
	MoveL Offs(p0,563.2,596.0, 0), v100, z5, tool0;
	MoveL Offs(p0,556.2,607.0, 0), v100, z5, tool0;
	MoveL Offs(p0,563.4,620.6, 0), v100, z5, tool0;
	MoveL Offs(p0,564.6028000000001,622.7674000000001, 0), v100, z5, tool0;
	MoveL Offs(p0,565.7984,624.8112000000002, 0), v100, z5, tool0;
	MoveL Offs(p0,566.9676000000001,626.7038, 0), v100, z5, tool0;
	MoveL Offs(p0,568.0912000000001,628.4176, 0), v100, z5, tool0;
	MoveL Offs(p0,569.15,629.925, 0), v100, z5, tool0;
	MoveL Offs(p0,570.1247999999999,631.1984, 0), v100, z5, tool0;
	MoveL Offs(p0,570.9964,632.2101999999999, 0), v100, z5, tool0;
	MoveL Offs(p0,571.7456,632.9328, 0), v100, z5, tool0;
	MoveL Offs(p0,572.3532,633.3386, 0), v100, z5, tool0;
	MoveL Offs(p0,572.8,633.4, 0), v100, z5, tool0;
	MoveL Offs(p0,574.9632,631.3872, 0), v100, z5, tool0;
	MoveL Offs(p0,575.675,630.425, 0), v100, z5, tool0;
	MoveL Offs(p0,576.4287999999999,629.3248, 0), v100, z5, tool0;
	MoveL Offs(p0,577.2113999999999,628.1094, 0), v100, z5, tool0;
	MoveL Offs(p0,578.0096,626.8016, 0), v100, z5, tool0;
	MoveL Offs(p0,578.8102000000001,625.4242, 0), v100, z5, tool0;
	MoveL Offs(p0,579.6,624.0, 0), v100, z5, tool0;
	MoveL Offs(p0,579.6,624.0, 0), v100, z5, tool0;
	MoveJ Offs(p0,101.6,606.8, 10), v100, z1, tool0;
	MoveL Offs(p0,103.3312,604.3872, 0), v100, z5, tool0;
	MoveL Offs(p0,103.875,603.55, 0), v100, z5, tool0;
	MoveL Offs(p0,104.43679999999999,602.6528, 0), v100, z5, tool0;
	MoveL Offs(p0,105.00340000000001,601.7124, 0), v100, z5, tool0;
	MoveL Offs(p0,105.5616,600.7456, 0), v100, z5, tool0;
	MoveL Offs(p0,106.09819999999999,599.7692, 0), v100, z5, tool0;
	MoveL Offs(p0,106.6,598.8, 0), v100, z5, tool0;
	MoveL Offs(p0,107.77920000000003,596.7856, 0), v100, z5, tool0;
	MoveL Offs(p0,108.26679999999999,596.0694, 0), v100, z5, tool0;
	MoveL Offs(p0,108.68960000000001,595.5488000000001, 0), v100, z5, tool0;
	MoveL Offs(p0,109.05,595.225, 0), v100, z5, tool0;
	MoveL Offs(p0,109.3504,595.0992, 0), v100, z5, tool0;
	MoveL Offs(p0,109.5932,595.1726, 0), v100, z5, tool0;
	MoveL Offs(p0,109.7808,595.4464, 0), v100, z5, tool0;
	MoveL Offs(p0,109.9156,595.9218000000001, 0), v100, z5, tool0;
	MoveL Offs(p0,110.0,596.6, 0), v100, z5, tool0;
	MoveL Offs(p0,110.40640000000003,599.1600000000001, 0), v100, z5, tool0;
	MoveL Offs(p0,110.88559999999998,599.768, 0), v100, z5, tool0;
	MoveL Offs(p0,111.52320000000002,599.9440000000001, 0), v100, z5, tool0;
	MoveL Offs(p0,112.3,599.7, 0), v100, z5, tool0;
	MoveL Offs(p0,113.19679999999998,599.048, 0), v100, z5, tool0;
	MoveL Offs(p0,114.1944,598.0, 0), v100, z5, tool0;
	MoveL Offs(p0,115.27360000000002,596.568, 0), v100, z5, tool0;
	MoveL Offs(p0,116.4152,594.7640000000001, 0), v100, z5, tool0;
	MoveL Offs(p0,117.6,592.6, 0), v100, z5, tool0;
	MoveL Offs(p0,119.75840000000001,587.9842000000001, 0), v100, z5, tool0;
	MoveL Offs(p0,121.57120000000005,583.4896000000001, 0), v100, z5, tool0;
	MoveL Offs(p0,123.06479999999999,578.9254, 0), v100, z5, tool0;
	MoveL Offs(p0,124.26560000000002,574.1008, 0), v100, z5, tool0;
	MoveL Offs(p0,125.2,568.825, 0), v100, z5, tool0;
	MoveL Offs(p0,125.89439999999999,562.9071999999999, 0), v100, z5, tool0;
	MoveL Offs(p0,126.37519999999999,556.1566, 0), v100, z5, tool0;
	MoveL Offs(p0,126.6688,548.3824000000001, 0), v100, z5, tool0;
	MoveL Offs(p0,126.80160000000001,539.3938, 0), v100, z5, tool0;
	MoveL Offs(p0,126.8,529.0, 0), v100, z5, tool0;
	MoveL Offs(p0,126.73020000000001,518.8848, 0), v100, z5, tool0;
	MoveL Offs(p0,126.5056,509.9024000000001, 0), v100, z5, tool0;
	MoveL Offs(p0,126.1034,501.8776, 0), v100, z5, tool0;
	MoveL Offs(p0,125.50080000000003,494.63520000000005, 0), v100, z5, tool0;
	MoveL Offs(p0,124.675,488.0, 0), v100, z5, tool0;
	MoveL Offs(p0,123.60320000000002,481.79679999999996, 0), v100, z5, tool0;
	MoveL Offs(p0,122.26259999999999,475.8503999999999, 0), v100, z5, tool0;
	MoveL Offs(p0,120.63040000000001,469.9856, 0), v100, z5, tool0;
	MoveL Offs(p0,118.68380000000002,464.0272000000001, 0), v100, z5, tool0;
	MoveL Offs(p0,116.4,457.8, 0), v100, z5, tool0;
	MoveL Offs(p0,114.2,452.4, 0), v100, z5, tool0;
	MoveL Offs(p0,103.6,456.6, 0), v100, z5, tool0;
	MoveL Offs(p0,100.31580000000002,457.8546000000001, 0), v100, z5, tool0;
	MoveL Offs(p0,97.75040000000003,458.90880000000016, 0), v100, z5, tool0;
	MoveL Offs(p0,95.85459999999999,460.0182000000001, 0), v100, z5, tool0;
	MoveL Offs(p0,94.5792,461.4384, 0), v100, z5, tool0;
	MoveL Offs(p0,93.875,463.425, 0), v100, z5, tool0;
	MoveL Offs(p0,93.6928,466.2336, 0), v100, z5, tool0;
	MoveL Offs(p0,93.98339999999999,470.11980000000005, 0), v100, z5, tool0;
	MoveL Offs(p0,94.69760000000001,475.33920000000006, 0), v100, z5, tool0;
	MoveL Offs(p0,95.78620000000001,482.1474, 0), v100, z5, tool0;
	MoveL Offs(p0,97.2,490.8, 0), v100, z5, tool0;
	MoveL Offs(p0,98.48,500.56359999999995, 0), v100, z5, tool0;
	MoveL Offs(p0,99.32800000000003,510.9728000000001, 0), v100, z5, tool0;
	MoveL Offs(p0,99.756,521.7852, 0), v100, z5, tool0;
	MoveL Offs(p0,99.77600000000001,532.7584, 0), v100, z5, tool0;
	MoveL Offs(p0,99.4,543.65, 0), v100, z5, tool0;
	MoveL Offs(p0,98.64,554.2176, 0), v100, z5, tool0;
	MoveL Offs(p0,97.508,564.2188, 0), v100, z5, tool0;
	MoveL Offs(p0,96.016,573.4112000000001, 0), v100, z5, tool0;
	MoveL Offs(p0,94.176,581.5524, 0), v100, z5, tool0;
	MoveL Offs(p0,92.0,588.4, 0), v100, z5, tool0;
	MoveL Offs(p0,91.24320000000003,590.4008000000001, 0), v100, z5, tool0;
	MoveL Offs(p0,90.64960000000004,592.0944000000002, 0), v100, z5, tool0;
	MoveL Offs(p0,90.2144,593.4975999999999, 0), v100, z5, tool0;
	MoveL Offs(p0,89.93280000000001,594.6272000000001, 0), v100, z5, tool0;
	MoveL Offs(p0,89.8,595.5, 0), v100, z5, tool0;
	MoveL Offs(p0,89.8112,596.1328, 0), v100, z5, tool0;
	MoveL Offs(p0,89.9616,596.5424, 0), v100, z5, tool0;
	MoveL Offs(p0,90.24640000000002,596.7456, 0), v100, z5, tool0;
	MoveL Offs(p0,90.66080000000001,596.7592000000001, 0), v100, z5, tool0;
	MoveL Offs(p0,91.2,596.6, 0), v100, z5, tool0;
	MoveL Offs(p0,93.01760000000002,594.4176000000001, 0), v100, z5, tool0;
	MoveL Offs(p0,92.9442,594.1052000000001, 0), v100, z5, tool0;
	MoveL Offs(p0,92.8,593.8, 0), v100, z5, tool0;
	MoveL Offs(p0,96.625,595.675, 0), v100, z5, tool0;
	MoveL Offs(p0,96.6736,596.5840000000001, 0), v100, z5, tool0;
	MoveL Offs(p0,96.61179999999999,597.673, 0), v100, z5, tool0;
	MoveL Offs(p0,96.4432,598.96, 0), v100, z5, tool0;
	MoveL Offs(p0,96.17139999999999,600.463, 0), v100, z5, tool0;
	MoveL Offs(p0,95.8,602.2, 0), v100, z5, tool0;
	MoveL Offs(p0,94.94800000000001,606.0070000000001, 0), v100, z5, tool0;
	MoveL Offs(p0,94.31200000000001,609.1600000000001, 0), v100, z5, tool0;
	MoveL Offs(p0,93.89200000000001,611.677, 0), v100, z5, tool0;
	MoveL Offs(p0,93.68800000000002,613.576, 0), v100, z5, tool0;
	MoveL Offs(p0,93.7,614.875, 0), v100, z5, tool0;
	MoveL Offs(p0,93.928,615.592, 0), v100, z5, tool0;
	MoveL Offs(p0,94.372,615.745, 0), v100, z5, tool0;
	MoveL Offs(p0,95.03200000000001,615.3520000000001, 0), v100, z5, tool0;
	MoveL Offs(p0,95.908,614.431, 0), v100, z5, tool0;
	MoveL Offs(p0,97.0,613.0, 0), v100, z5, tool0;
	MoveL Offs(p0,98.5102,610.9174, 0), v100, z5, tool0;
	MoveL Offs(p0,99.0224,610.2128, 0), v100, z5, tool0;
	MoveL Offs(p0,99.525,609.525, 0), v100, z5, tool0;
	MoveL Offs(p0,100.0096,608.8672, 0), v100, z5, tool0;
	MoveL Offs(p0,100.4678,608.2526, 0), v100, z5, tool0;
	MoveL Offs(p0,100.8912,607.6944000000001, 0), v100, z5, tool0;
	MoveL Offs(p0,101.2714,607.2058, 0), v100, z5, tool0;
	MoveL Offs(p0,101.6,606.8, 0), v100, z5, tool0;
	MoveL Offs(p0,101.6,606.8, 0), v100, z5, tool0;
	MoveJ Offs(p0,787.8,603.6, 10), v100, z1, tool0;
	MoveL Offs(p0,785.3724000000001,600.9768000000001, 0), v100, z5, tool0;
	MoveL Offs(p0,783.1392000000003,598.1664000000003, 0), v100, z5, tool0;
	MoveL Offs(p0,781.1148000000001,595.1976, 0), v100, z5, tool0;
	MoveL Offs(p0,779.3136000000001,592.0992, 0), v100, z5, tool0;
	MoveL Offs(p0,777.75,588.9, 0), v100, z5, tool0;
	MoveL Offs(p0,776.4384,585.6288, 0), v100, z5, tool0;
	MoveL Offs(p0,775.3932,582.3144, 0), v100, z5, tool0;
	MoveL Offs(p0,774.6288000000001,578.9856, 0), v100, z5, tool0;
	MoveL Offs(p0,774.1596000000001,575.6712, 0), v100, z5, tool0;
	MoveL Offs(p0,774.0,572.4, 0), v100, z5, tool0;
	MoveL Offs(p0,774.1046000000001,569.3824000000001, 0), v100, z5, tool0;
	MoveL Offs(p0,774.4288000000003,566.5472000000002, 0), v100, z5, tool0;
	MoveL Offs(p0,774.9882,563.8608, 0), v100, z5, tool0;
	MoveL Offs(p0,775.7984,561.2896000000001, 0), v100, z5, tool0;
	MoveL Offs(p0,776.875,558.8, 0), v100, z5, tool0;
	MoveL Offs(p0,778.2336,556.3583999999998, 0), v100, z5, tool0;
	MoveL Offs(p0,779.8897999999999,553.9312, 0), v100, z5, tool0;
	MoveL Offs(p0,781.8592000000001,551.4848, 0), v100, z5, tool0;
	MoveL Offs(p0,784.1574,548.9856, 0), v100, z5, tool0;
	MoveL Offs(p0,786.8,546.4, 0), v100, z5, tool0;
	MoveL Offs(p0,788.9960000000002,544.1656, 0), v100, z5, tool0;
	MoveL Offs(p0,790.7840000000002,542.0128000000002, 0), v100, z5, tool0;
	MoveL Offs(p0,792.164,539.9272000000001, 0), v100, z5, tool0;
	MoveL Offs(p0,793.1360000000001,537.8944, 0), v100, z5, tool0;
	MoveL Offs(p0,793.7,535.9, 0), v100, z5, tool0;
	MoveL Offs(p0,793.856,533.9296, 0), v100, z5, tool0;
	MoveL Offs(p0,793.6039999999999,531.9688, 0), v100, z5, tool0;
	MoveL Offs(p0,792.9440000000001,530.0032000000001, 0), v100, z5, tool0;
	MoveL Offs(p0,791.876,528.0184, 0), v100, z5, tool0;
	MoveL Offs(p0,790.4,526.0, 0), v100, z5, tool0;
	MoveL Offs(p0,788.2752000000003,523.9248000000001, 0), v100, z5, tool0;
	MoveL Offs(p0,786.8108,523.1812, 0), v100, z5, tool0;
	MoveL Offs(p0,784.7776000000001,522.5984000000001, 0), v100, z5, tool0;
	MoveL Offs(p0,781.95,522.15, 0), v100, z5, tool0;
	MoveL Offs(p0,778.1024,521.8095999999999, 0), v100, z5, tool0;
	MoveL Offs(p0,773.0092000000001,521.5508, 0), v100, z5, tool0;
	MoveL Offs(p0,766.4448,521.3471999999999, 0), v100, z5, tool0;
	MoveL Offs(p0,758.1836000000001,521.1724, 0), v100, z5, tool0;
	MoveL Offs(p0,748.0,521.0, 0), v100, z5, tool0;
	MoveL Offs(p0,738.9566000000002,520.8714000000001, 0), v100, z5, tool0;
	MoveL Offs(p0,731.1648000000002,520.7152000000002, 0), v100, z5, tool0;
	MoveL Offs(p0,724.4721999999999,520.5157999999999, 0), v100, z5, tool0;
	MoveL Offs(p0,718.7264,520.2576, 0), v100, z5, tool0;
	MoveL Offs(p0,713.775,519.925, 0), v100, z5, tool0;
	MoveL Offs(p0,709.4656000000001,519.5024000000001, 0), v100, z5, tool0;
	MoveL Offs(p0,705.6458,518.9741999999999, 0), v100, z5, tool0;
	MoveL Offs(p0,702.1632000000001,518.3248000000001, 0), v100, z5, tool0;
	MoveL Offs(p0,698.8654,517.5386000000001, 0), v100, z5, tool0;
	MoveL Offs(p0,695.6,516.6, 0), v100, z5, tool0;
	MoveL Offs(p0,693.3724000000001,515.9770000000001, 0), v100, z5, tool0;
	MoveL Offs(p0,691.2672000000002,515.4320000000001, 0), v100, z5, tool0;
	MoveL Offs(p0,689.3108,514.971, 0), v100, z5, tool0;
	MoveL Offs(p0,687.5296000000001,514.6, 0), v100, z5, tool0;
	MoveL Offs(p0,685.95,514.325, 0), v100, z5, tool0;
	MoveL Offs(p0,684.5984,514.152, 0), v100, z5, tool0;
	MoveL Offs(p0,683.5012,514.087, 0), v100, z5, tool0;
	MoveL Offs(p0,682.6848000000001,514.1360000000001, 0), v100, z5, tool0;
	MoveL Offs(p0,682.1756,514.3050000000001, 0), v100, z5, tool0;
	MoveL Offs(p0,682.0,514.6, 0), v100, z5, tool0;
	MoveL Offs(p0,683.1447999999999,517.4224, 0), v100, z5, tool0;
	MoveL Offs(p0,683.9776,519.1088, 0), v100, z5, tool0;
	MoveL Offs(p0,685.0,521.1, 0), v100, z5, tool0;
	MoveL Offs(p0,686.1904,523.3552, 0), v100, z5, tool0;
	MoveL Offs(p0,687.5271999999999,525.8335999999999, 0), v100, z5, tool0;
	MoveL Offs(p0,688.9888000000001,528.4944000000002, 0), v100, z5, tool0;
	MoveL Offs(p0,690.5536,531.2968000000001, 0), v100, z5, tool0;
	MoveL Offs(p0,692.2,534.2, 0), v100, z5, tool0;
	MoveL Offs(p0,694.5202000000002,538.2360000000001, 0), v100, z5, tool0;
	MoveL Offs(p0,696.4576000000003,541.7440000000001, 0), v100, z5, tool0;
	MoveL Offs(p0,698.0374,544.784, 0), v100, z5, tool0;
	MoveL Offs(p0,699.2848000000001,547.4159999999999, 0), v100, z5, tool0;
	MoveL Offs(p0,700.225,549.7, 0), v100, z5, tool0;
	MoveL Offs(p0,700.8832,551.696, 0), v100, z5, tool0;
	MoveL Offs(p0,701.2846,553.464, 0), v100, z5, tool0;
	MoveL Offs(p0,701.4544,555.0640000000001, 0), v100, z5, tool0;
	MoveL Offs(p0,701.4177999999999,556.556, 0), v100, z5, tool0;
	MoveL Offs(p0,701.2,558.0, 0), v100, z5, tool0;
	MoveL Offs(p0,700.8640000000003,560.8304000000002, 0), v100, z5, tool0;
	MoveL Offs(p0,700.948,562.0175999999999, 0), v100, z5, tool0;
	MoveL Offs(p0,701.248,563.1232000000001, 0), v100, z5, tool0;
	MoveL Offs(p0,701.8,564.2, 0), v100, z5, tool0;
	MoveL Offs(p0,702.64,565.3008, 0), v100, z5, tool0;
	MoveL Offs(p0,703.804,566.4784, 0), v100, z5, tool0;
	MoveL Offs(p0,705.3280000000001,567.7856, 0), v100, z5, tool0;
	MoveL Offs(p0,707.2479999999999,569.2751999999999, 0), v100, z5, tool0;
	MoveL Offs(p0,709.6,571.0, 0), v100, z5, tool0;
	MoveL Offs(p0,713.755,573.8994, 0), v100, z5, tool0;
	MoveL Offs(p0,718.6960000000001,577.0352, 0), v100, z5, tool0;
	MoveL Offs(p0,724.2969999999999,580.3438, 0), v100, z5, tool0;
	MoveL Offs(p0,730.432,583.7616, 0), v100, z5, tool0;
	MoveL Offs(p0,736.975,587.225, 0), v100, z5, tool0;
	MoveL Offs(p0,743.8,590.6704, 0), v100, z5, tool0;
	MoveL Offs(p0,750.781,594.0342, 0), v100, z5, tool0;
	MoveL Offs(p0,757.792,597.2528, 0), v100, z5, tool0;
	MoveL Offs(p0,764.707,600.2626, 0), v100, z5, tool0;
	MoveL Offs(p0,771.4,603.0, 0), v100, z5, tool0;
	MoveL Offs(p0,777.4266,605.3226000000001, 0), v100, z5, tool0;
	MoveL Offs(p0,782.3408000000002,607.1328000000001, 0), v100, z5, tool0;
	MoveL Offs(p0,786.1942,608.4341999999999, 0), v100, z5, tool0;
	MoveL Offs(p0,789.0384,609.2304000000001, 0), v100, z5, tool0;
	MoveL Offs(p0,790.925,609.525, 0), v100, z5, tool0;
	MoveL Offs(p0,791.9056,609.3216, 0), v100, z5, tool0;
	MoveL Offs(p0,792.0318,608.6238, 0), v100, z5, tool0;
	MoveL Offs(p0,791.3552000000001,607.4352000000001, 0), v100, z5, tool0;
	MoveL Offs(p0,789.9274,605.7594000000001, 0), v100, z5, tool0;
	MoveL Offs(p0,787.8,603.6, 0), v100, z5, tool0;
	MoveL Offs(p0,787.8,603.6, 0), v100, z5, tool0;
	MoveJ Offs(p0,50.8,529.2, 10), v100, z1, tool0;
	MoveL Offs(p0,53.618200000000016,523.3618, 0), v100, z5, tool0;
	MoveL Offs(p0,56.641600000000004,517.5344000000002, 0), v100, z5, tool0;
	MoveL Offs(p0,59.82340000000001,511.7886, 0), v100, z5, tool0;
	MoveL Offs(p0,63.1168,506.1952000000001, 0), v100, z5, tool0;
	MoveL Offs(p0,66.475,500.825, 0), v100, z5, tool0;
	MoveL Offs(p0,69.8512,495.7488, 0), v100, z5, tool0;
	MoveL Offs(p0,73.1986,491.0374, 0), v100, z5, tool0;
	MoveL Offs(p0,76.47040000000001,486.7616, 0), v100, z5, tool0;
	MoveL Offs(p0,79.61980000000001,482.9922, 0), v100, z5, tool0;
	MoveL Offs(p0,82.6,479.8, 0), v100, z5, tool0;
	MoveL Offs(p0,84.75900000000001,477.48240000000015, 0), v100, z5, tool0;
	MoveL Offs(p0,86.55200000000004,475.2272000000001, 0), v100, z5, tool0;
	MoveL Offs(p0,87.973,473.0607999999999, 0), v100, z5, tool0;
	MoveL Offs(p0,89.016,471.00960000000015, 0), v100, z5, tool0;
	MoveL Offs(p0,89.675,469.1, 0), v100, z5, tool0;
	MoveL Offs(p0,89.94399999999999,467.35839999999996, 0), v100, z5, tool0;
	MoveL Offs(p0,89.817,465.81119999999993, 0), v100, z5, tool0;
	MoveL Offs(p0,89.28800000000001,464.4848, 0), v100, z5, tool0;
	MoveL Offs(p0,88.35100000000001,463.40560000000005, 0), v100, z5, tool0;
	MoveL Offs(p0,87.0,462.6, 0), v100, z5, tool0;
	MoveL Offs(p0,84.62720000000003,462.7008000000002, 0), v100, z5, tool0;
	MoveL Offs(p0,83.21279999999999,463.2012, 0), v100, z5, tool0;
	MoveL Offs(p0,81.7456,463.9344000000001, 0), v100, z5, tool0;
	MoveL Offs(p0,80.3,464.85, 0), v100, z5, tool0;
	MoveL Offs(p0,78.95039999999999,465.89759999999995, 0), v100, z5, tool0;
	MoveL Offs(p0,77.7712,467.0268, 0), v100, z5, tool0;
	MoveL Offs(p0,76.83680000000001,468.18720000000013, 0), v100, z5, tool0;
	MoveL Offs(p0,76.2216,469.3284, 0), v100, z5, tool0;
	MoveL Offs(p0,76.0,470.4, 0), v100, z5, tool0;
	MoveL Offs(p0,74.5216,473.5488, 0), v100, z5, tool0;
	MoveL Offs(p0,73.75,474.9, 0), v100, z5, tool0;
	MoveL Offs(p0,72.84639999999999,476.41919999999993, 0), v100, z5, tool0;
	MoveL Offs(p0,71.8252,478.07759999999996, 0), v100, z5, tool0;
	MoveL Offs(p0,70.7008,479.8464, 0), v100, z5, tool0;
	MoveL Offs(p0,69.4876,481.6968, 0), v100, z5, tool0;
	MoveL Offs(p0,68.2,483.6, 0), v100, z5, tool0;
	MoveL Offs(p0,63.5172,490.79180000000014, 0), v100, z5, tool0;
	MoveL Offs(p0,59.081600000000016,498.2944000000001, 0), v100, z5, tool0;
	MoveL Offs(p0,54.91239999999999,506.0586, 0), v100, z5, tool0;
	MoveL Offs(p0,51.028800000000004,514.0352, 0), v100, z5, tool0;
	MoveL Offs(p0,47.45,522.175, 0), v100, z5, tool0;
	MoveL Offs(p0,44.1952,530.4288, 0), v100, z5, tool0;
	MoveL Offs(p0,41.2836,538.7474, 0), v100, z5, tool0;
	MoveL Offs(p0,38.73440000000001,547.0816000000001, 0), v100, z5, tool0;
	MoveL Offs(p0,36.5668,555.3822, 0), v100, z5, tool0;
	MoveL Offs(p0,34.8,563.6, 0), v100, z5, tool0;
	MoveL Offs(p0,33.555600000000005,570.3480000000001, 0), v100, z5, tool0;
	MoveL Offs(p0,32.69280000000001,575.7040000000002, 0), v100, z5, tool0;
	MoveL Offs(p0,32.1972,579.656, 0), v100, z5, tool0;
	MoveL Offs(p0,32.0544,582.1920000000001, 0), v100, z5, tool0;
	MoveL Offs(p0,32.25,583.3, 0), v100, z5, tool0;
	MoveL Offs(p0,32.769600000000004,582.9680000000001, 0), v100, z5, tool0;
	MoveL Offs(p0,33.5988,581.184, 0), v100, z5, tool0;
	MoveL Offs(p0,34.723200000000006,577.936, 0), v100, z5, tool0;
	MoveL Offs(p0,36.1284,573.212, 0), v100, z5, tool0;
	MoveL Offs(p0,37.8,567.0, 0), v100, z5, tool0;
	MoveL Offs(p0,38.833600000000004,563.2632000000001, 0), v100, z5, tool0;
	MoveL Offs(p0,39.996800000000015,559.3056000000003, 0), v100, z5, tool0;
	MoveL Offs(p0,41.2632,555.2064, 0), v100, z5, tool0;
	MoveL Offs(p0,42.6064,551.0448, 0), v100, z5, tool0;
	MoveL Offs(p0,44.0,546.9, 0), v100, z5, tool0;
	MoveL Offs(p0,45.41760000000001,542.8511999999998, 0), v100, z5, tool0;
	MoveL Offs(p0,46.8328,538.9775999999999, 0), v100, z5, tool0;
	MoveL Offs(p0,48.21920000000001,535.3584000000001, 0), v100, z5, tool0;
	MoveL Offs(p0,49.5504,532.0728, 0), v100, z5, tool0;
	MoveL Offs(p0,50.8,529.2, 0), v100, z5, tool0;
	MoveL Offs(p0,50.8,529.2, 0), v100, z5, tool0;
	MoveJ Offs(p0,72.6,578.0, 10), v100, z1, tool0;
	MoveL Offs(p0,76.6,584.4, 0), v100, z5, tool0;
	MoveL Offs(p0,80.6,576.8, 0), v100, z5, tool0;
	MoveL Offs(p0,84.4,569.2, 0), v100, z5, tool0;
	MoveL Offs(p0,88.0,573.8, 0), v100, z5, tool0;
	MoveL Offs(p0,89.59520000000003,575.9200000000002, 0), v100, z5, tool0;
	MoveL Offs(p0,90.1888,576.5989999999999, 0), v100, z5, tool0;
	MoveL Offs(p0,90.6816,577.032, 0), v100, z5, tool0;
	MoveL Offs(p0,91.1,577.225, 0), v100, z5, tool0;
	MoveL Offs(p0,91.4704,577.184, 0), v100, z5, tool0;
	MoveL Offs(p0,91.8192,576.915, 0), v100, z5, tool0;
	MoveL Offs(p0,92.17280000000001,576.424, 0), v100, z5, tool0;
	MoveL Offs(p0,92.55760000000001,575.717, 0), v100, z5, tool0;
	MoveL Offs(p0,93.0,574.8, 0), v100, z5, tool0;
	MoveL Offs(p0,93.77860000000001,571.4534000000001, 0), v100, z5, tool0;
	MoveL Offs(p0,94.42880000000002,565.9312000000001, 0), v100, z5, tool0;
	MoveL Offs(p0,94.94219999999999,558.7098, 0), v100, z5, tool0;
	MoveL Offs(p0,95.31039999999999,550.2656, 0), v100, z5, tool0;
	MoveL Offs(p0,95.525,541.075, 0), v100, z5, tool0;
	MoveL Offs(p0,95.57759999999999,531.6144, 0), v100, z5, tool0;
	MoveL Offs(p0,95.4598,522.3602000000001, 0), v100, z5, tool0;
	MoveL Offs(p0,95.1632,513.7888, 0), v100, z5, tool0;
	MoveL Offs(p0,94.67940000000002,506.37659999999994, 0), v100, z5, tool0;
	MoveL Offs(p0,94.0,500.6, 0), v100, z5, tool0;
	MoveL Offs(p0,93.07160000000002,494.81139999999994, 0), v100, z5, tool0;
	MoveL Offs(p0,92.28480000000002,490.2192000000001, 0), v100, z5, tool0;
	MoveL Offs(p0,91.57719999999999,486.7237999999999, 0), v100, z5, tool0;
	MoveL Offs(p0,90.88640000000001,484.22560000000004, 0), v100, z5, tool0;
	MoveL Offs(p0,90.15,482.625, 0), v100, z5, tool0;
	MoveL Offs(p0,89.3056,481.8224, 0), v100, z5, tool0;
	MoveL Offs(p0,88.29079999999999,481.71819999999997, 0), v100, z5, tool0;
	MoveL Offs(p0,87.0432,482.2128000000001, 0), v100, z5, tool0;
	MoveL Offs(p0,85.5004,483.2066, 0), v100, z5, tool0;
	MoveL Offs(p0,83.6,484.6, 0), v100, z5, tool0;
	MoveL Offs(p0,79.2586,488.74680000000006, 0), v100, z5, tool0;
	MoveL Offs(p0,74.30880000000002,495.1184000000001, 0), v100, z5, tool0;
	MoveL Offs(p0,68.9822,503.25159999999994, 0), v100, z5, tool0;
	MoveL Offs(p0,63.510400000000004,512.6832, 0), v100, z5, tool0;
	MoveL Offs(p0,58.125,522.95, 0), v100, z5, tool0;
	MoveL Offs(p0,53.057599999999994,533.5887999999999, 0), v100, z5, tool0;
	MoveL Offs(p0,48.5398,544.1364, 0), v100, z5, tool0;
	MoveL Offs(p0,44.803200000000004,554.1296, 0), v100, z5, tool0;
	MoveL Offs(p0,42.0794,563.1052000000001, 0), v100, z5, tool0;
	MoveL Offs(p0,40.6,570.6, 0), v100, z5, tool0;
	MoveL Offs(p0,40.29380000000001,573.558, 0), v100, z5, tool0;
	MoveL Offs(p0,40.21440000000001,575.9520000000001, 0), v100, z5, tool0;
	MoveL Offs(p0,40.360600000000005,577.7819999999999, 0), v100, z5, tool0;
	MoveL Offs(p0,40.73120000000001,579.048, 0), v100, z5, tool0;
	MoveL Offs(p0,41.325,579.75, 0), v100, z5, tool0;
	MoveL Offs(p0,42.1408,579.8879999999999, 0), v100, z5, tool0;
	MoveL Offs(p0,43.1774,579.462, 0), v100, z5, tool0;
	MoveL Offs(p0,44.4336,578.472, 0), v100, z5, tool0;
	MoveL Offs(p0,45.9082,576.918, 0), v100, z5, tool0;
	MoveL Offs(p0,47.6,574.8, 0), v100, z5, tool0;
	MoveL Offs(p0,51.4,569.4, 0), v100, z5, tool0;
	MoveL Offs(p0,56.0,577.0, 0), v100, z5, tool0;
	MoveL Offs(p0,60.6,584.4, 0), v100, z5, tool0;
	MoveL Offs(p0,64.6,578.0, 0), v100, z5, tool0;
	MoveL Offs(p0,68.6,571.6, 0), v100, z5, tool0;
	MoveL Offs(p0,72.6,578.0, 0), v100, z5, tool0;
	MoveL Offs(p0,72.6,578.0, 0), v100, z5, tool0;
	MoveJ Offs(p0,173.4,565.6, 10), v100, z1, tool0;
	MoveL Offs(p0,172.377,554.975, 0), v100, z5, tool0;
	MoveL Offs(p0,170.66400000000004,544.0800000000002, 0), v100, z5, tool0;
	MoveL Offs(p0,168.315,533.0649999999999, 0), v100, z5, tool0;
	MoveL Offs(p0,165.384,522.08, 0), v100, z5, tool0;
	MoveL Offs(p0,161.925,511.275, 0), v100, z5, tool0;
	MoveL Offs(p0,157.99200000000002,500.8, 0), v100, z5, tool0;
	MoveL Offs(p0,153.63899999999998,490.805, 0), v100, z5, tool0;
	MoveL Offs(p0,148.92000000000002,481.44000000000005, 0), v100, z5, tool0;
	MoveL Offs(p0,143.889,472.855, 0), v100, z5, tool0;
	MoveL Offs(p0,138.6,465.2, 0), v100, z5, tool0;
	MoveL Offs(p0,136.8938,462.9434000000001, 0), v100, z5, tool0;
	MoveL Offs(p0,135.27040000000005,460.7552000000002, 0), v100, z5, tool0;
	MoveL Offs(p0,133.75259999999997,458.6678, 0), v100, z5, tool0;
	MoveL Offs(p0,132.3632,456.71359999999993, 0), v100, z5, tool0;
	MoveL Offs(p0,131.125,454.925, 0), v100, z5, tool0;
	MoveL Offs(p0,130.06080000000003,453.3344, 0), v100, z5, tool0;
	MoveL Offs(p0,129.1934,451.9742, 0), v100, z5, tool0;
	MoveL Offs(p0,128.5456,450.8768, 0), v100, z5, tool0;
	MoveL Offs(p0,128.1402,450.07460000000003, 0), v100, z5, tool0;
	MoveL Offs(p0,128.0,449.6, 0), v100, z5, tool0;
	MoveL Offs(p0,125.9028,448.1944, 0), v100, z5, tool0;
	MoveL Offs(p0,125.3632,448.0896000000001, 0), v100, z5, tool0;
	MoveL Offs(p0,124.7924,448.0232, 0), v100, z5, tool0;
	MoveL Offs(p0,124.2,448.0, 0), v100, z5, tool0;
	MoveL Offs(p0,121.7844,448.3348, 0), v100, z5, tool0;
	MoveL Offs(p0,121.41280000000002,448.7296, 0), v100, z5, tool0;
	MoveL Offs(p0,121.25,449.35, 0), v100, z5, tool0;
	MoveL Offs(p0,121.2912,450.2464, 0), v100, z5, tool0;
	MoveL Offs(p0,121.5316,451.4692, 0), v100, z5, tool0;
	MoveL Offs(p0,121.96640000000002,453.0688, 0), v100, z5, tool0;
	MoveL Offs(p0,122.59080000000002,455.0956, 0), v100, z5, tool0;
	MoveL Offs(p0,123.4,457.6, 0), v100, z5, tool0;
	MoveL Offs(p0,124.74400000000003,460.9376000000001, 0), v100, z5, tool0;
	MoveL Offs(p0,125.58699999999999,462.7174, 0), v100, z5, tool0;
